LIN {X 0,Y 260.19,Z 606.09,A -85,B 0,C 180,E1 -26180.673,E2 -26180.673} C_VEL
LIN {X 0,Y 265.436,Z 608.192,A -85,B 0,C 180,E1 -26182.392,E2 -26182.392} C_VEL
LIN {X 0,Y 269.491,Z 609.865,A -85,B 0,C 180,E1 -26184.012,E2 -26184.012} C_VEL
LIN {X 0,Y 272.352,Z 611.178,A -85,B 0,C 180,E1 -26185.56,E2 -26185.56} C_VEL
LIN {X 0,Y 274.974,Z 612.087,A -85,B 0,C 180,E1 -26187.07,E2 -26187.07} C_VEL
LIN {X 0,Y 276.592,Z 612.646,A -85,B 0,C 180,E1 -26188.544,E2 -26188.544} C_VEL
LIN {X 0,Y 277.503,Z 612.825,A -85,B 0,C 180,E1 -26190,E2 -26190} C_VEL
LIN {X 0,Y 276.602,Z 612.645,A -85,B 0,C 180,E1 -26191.455,E2 -26191.455} C_VEL
LIN {X 0,Y 274.515,Z 611.947,A -85,B 0,C 180,E1 -26193.199,E2 -26193.199} C_VEL
LIN {X 0,Y 272.336,Z 611.179,A -85,B 0,C 180,E1 -26194.44,E2 -26194.44} C_VEL
LIN {X 0,Y 268.698,Z 609.555,A -85,B 0,C 180,E1 -26196.331,E2 -26196.331} C_VEL
LIN {X 0,Y 265.447,Z 608.193,A -85,B 0,C 180,E1 -26197.607,E2 -26197.607} C_VEL
LIN {X 0,Y 260.192,Z 606.091,A -85,B 0,C 180,E1 -26199.326,E2 -26199.326} C_VEL
LIN {X 0,Y 253.891,Z 603.535,A -85,B 0,C 180,E1 -26201.172,E2 -26201.172} C_VEL
LIN {X 0,Y 245.622,Z 600.226,A -85,B 0,C 180,E1 -26203.388,E2 -26203.388} C_VEL
LIN {X 0,Y 234.391,Z 595.435,A -85,B 0,C 180,E1 -26206.368,E2 -26206.368} C_VEL
LIN {X 0,Y 220.959,Z 588.75,A -85,B 0,C 180,E1 -26210.238,E2 -26210.238} C_VEL
LIN {X 0,Y 208.557,Z 580.602,A -85,B 0,C 180,E1 -26214.518,E2 -26214.518} C_VEL
LIN {X 0,Y 199.491,Z 572.681,A -85,B 0,C 180,E1 -26218.271,E2 -26218.271} C_VEL
LIN {X 0,Y 191.268,Z 563.212,A -85,B 0,C 180,E1 -26222.318,E2 -26222.318} C_VEL
LIN {X 0,Y 184.44,Z 553.289,A -85,B 0,C 180,E1 -26226.147,E2 -26226.147} C_VEL
LIN {X 0,Y 179.392,Z 544.208,A -85,B 0,C 180,E1 -26229.311,E2 -26229.311} C_VEL
LIN {X 0,Y 175.265,Z 535.205,A -85,B 0,C 180,E1 -26232.114,E2 -26232.114} C_VEL
LIN {X 0,Y 171.108,Z 524.747,A -85,B 0,C 180,E1 -26234.991,E2 -26234.991} C_VEL
LIN {X 0,Y 167.297,Z 514.145,A -85,B 0,C 180,E1 -26237.566,E2 -26237.566} C_VEL
LIN {X 0,Y 160.835,Z 495.6,A -85,B 0,C 180,E1 -26241.588,E2 -26241.588} C_VEL
LIN {X 0,Y 157.196,Z 486.8,A -85,B 0,C 180,E1 -26243.972,E2 -26243.972} C_VEL
LIN {X 0,Y 152.993,Z 478.107,A -85,B 0,C 180,E1 -26246.943,E2 -26246.943} C_VEL
LIN {X 0,Y 148.523,Z 469.896,A -85,B 0,C 180,E1 -26250.502,E2 -26250.502} C_VEL
LIN {X 0,Y 144.159,Z 462.807,A -85,B 0,C 180,E1 -26254.558,E2 -26254.558} C_VEL
LIN {X 0,Y 141.726,Z 459.081,A -85,B 0,C 180,E1 -26257.208,E2 -26257.208} C_VEL
LIN {X 0,Y 138.793,Z 454.797,A -85,B 0,C 180,E1 -26260.984,E2 -26260.984} C_VEL
LIN {X 0,Y 136.479,Z 451.612,A -85,B 0,C 180,E1 -26264.699,E2 -26264.699} C_VEL
LIN {X 0,Y 135.908,Z 450.393,A -85,B 0,C 180,E1 -26265.878,E2 -26265.878} C_VEL
LIN {X 0,Y 133.785,Z 448.176,A -85,B 0,C 180,E1 -26270.934,E2 -26270.934} C_VEL
LIN {X 0,Y 132.733,Z 445.405,A -85,B 0,C 180,E1 -26276.587,E2 -26276.587} C_VEL
LIN {X 0,Y 132.581,Z 444.946,A -85,B 0,C 180,E1 -26280.002,E2 -26280.002} C_VEL
LIN {X 0,Y 132.86,Z 445.806,A -85,B 0,C 180,E1 -26284.173,E2 -26284.173} C_VEL
LIN {X 0,Y 135.26,Z 449.966,A -85,B 0,C 180,E1 -26292.482,E2 -26292.482} C_VEL
LIN {X 0,Y 136.045,Z 450.627,A -85,B 0,C 180,E1 -26294.015,E2 -26294.015} C_VEL
LIN {X 0,Y 138.067,Z 454.011,A -85,B 0,C 180,E1 -26297.594,E2 -26297.594} C_VEL
LIN {X 0,Y 139.483,Z 455.822,A -85,B 0,C 180,E1 -26299.597,E2 -26299.597} C_VEL
LIN {X 0,Y 142.535,Z 460.338,A -85,B 0,C 180,E1 -26303.33,E2 -26303.33} C_VEL
LIN {X 0,Y 145.461,Z 464.955,A -85,B 0,C 180,E1 -26306.355,E2 -26306.355} C_VEL
LIN {X 0,Y 147.881,Z 468.942,A -85,B 0,C 180,E1 -26308.571,E2 -26308.571} C_VEL
LIN {X 0,Y 151.068,Z 476.333,A -85,B 0,C 180,E1 -26311.365,E2 -26311.365} C_VEL
LIN {X 0,Y 155.214,Z 487.342,A -85,B 0,C 180,E1 -26314.658,E2 -26314.658} C_VEL
LIN {X 0,Y 156.571,Z 491.711,A -85,B 0,C 180,E1 -26315.701,E2 -26315.701} C_VEL
LIN {X 0,Y 154.226,Z 518.872,A -85,B 0,C 180,E1 -26316.735,E2 -26316.735} C_VEL
LIN {X 0,Y 152.512,Z 529.749,A -85,B 0,C 180,E1 -26317.377,E2 -26317.377} C_VEL
LIN {X 0,Y 150.32,Z 539.537,A -85,B 0,C 180,E1 -26318.185,E2 -26318.185} C_VEL
LIN {X 0,Y 147.435,Z 549.33,A -85,B 0,C 180,E1 -26319.232,E2 -26319.232} C_VEL
LIN {X 0,Y 144.317,Z 558.091,A -85,B 0,C 180,E1 -26320.458,E2 -26320.458} C_VEL
LIN {X 0,Y 140.709,Z 566.811,A -85,B 0,C 180,E1 -26322.018,E2 -26322.018} C_VEL
LIN {X 0,Y 136.625,Z 575.317,A -85,B 0,C 180,E1 -26323.934,E2 -26323.934} C_VEL
LIN {X 0,Y 132.189,Z 583.484,A -85,B 0,C 180,E1 -26326.28,E2 -26326.28} C_VEL
LIN {X 0,Y 128.035,Z 590.426,A -85,B 0,C 180,E1 -26328.802,E2 -26328.802} C_VEL
LIN {X 0,Y 124.132,Z 596.412,A -85,B 0,C 180,E1 -26331.482,E2 -26331.482} C_VEL
LIN {X 0,Y 119.301,Z 603.383,A -85,B 0,C 180,E1 -26335.565,E2 -26335.565} C_VEL
LIN {X 0,Y 115.991,Z 608.001,A -85,B 0,C 180,E1 -26339.003,E2 -26339.003} C_VEL
LIN {X 0,Y 111.975,Z 613.094,A -85,B 0,C 180,E1 -26343.939,E2 -26343.939} C_VEL
LIN {X 0,Y 108.807,Z 617.061,A -85,B 0,C 180,E1 -26349.193,E2 -26349.193} C_VEL
LIN {X 0,Y 106.705,Z 620.004,A -85,B 0,C 180,E1 -26354.726,E2 -26354.726} C_VEL
LIN {X 0,Y 105.799,Z 621.512,A -85,B 0,C 180,E1 -26358.506,E2 -26358.506} C_VEL
LIN {X 0,Y 105.048,Z 623.051,A -85,B 0,C 180,E1 -26366.165,E2 -26366.165} C_VEL
LIN {X 0,Y 105.171,Z 623.337,A -85,B 0,C 180,E1 -26370.001,E2 -26370.001} C_VEL
LIN {X 0,Y 105.226,Z 622.446,A -85,B 0,C 180,E1 -26377.678,E2 -26377.678} C_VEL
LIN {X 0,Y 105.782,Z 621.511,A -85,B 0,C 180,E1 -26381.498,E2 -26381.498} C_VEL
LIN {X 0,Y 107.976,Z 618.15,A -85,B 0,C 180,E1 -26388.993,E2 -26388.993} C_VEL
LIN {X 0,Y 110.812,Z 614.521,A -85,B 0,C 180,E1 -26394.347,E2 -26394.347} C_VEL
LIN {X 0,Y 114.51,Z 609.787,A -85,B 0,C 180,E1 -26399.407,E2 -26399.407} C_VEL
LIN {X 0,Y 118.573,Z 604.41,A -85,B 0,C 180,E1 -26403.712,E2 -26403.712} C_VEL
LIN {X 0,Y 122.385,Z 599.035,A -85,B 0,C 180,E1 -26407.083,E2 -26407.083} C_VEL
LIN {X 0,Y 126.08,Z 593.543,A -85,B 0,C 180,E1 -26409.87,E2 -26409.87} C_VEL
LIN {X 0,Y 131.164,Z 585.33,A -85,B 0,C 180,E1 -26413.092,E2 -26413.092} C_VEL
LIN {X 0,Y 135.503,Z 577.507,A -85,B 0,C 180,E1 -26415.493,E2 -26415.493} C_VEL
LIN {X 0,Y 139.53,Z 569.429,A -85,B 0,C 180,E1 -26417.447,E2 -26417.447} C_VEL
LIN {X 0,Y 143.712,Z 559.673,A -85,B 0,C 180,E1 -26419.289,E2 -26419.289} C_VEL
LIN {X 0,Y 146.801,Z 551.287,A -85,B 0,C 180,E1 -26420.532,E2 -26420.532} C_VEL
LIN {X 0,Y 149.987,Z 540.786,A -85,B 0,C 180,E1 -26421.708,E2 -26421.708} C_VEL
LIN {X 0,Y 152.454,Z 530.424,A -85,B 0,C 180,E1 -26422.545,E2 -26422.545} C_VEL
LIN {X 0,Y 154.051,Z 520.443,A -85,B 0,C 180,E1 -26423.174,E2 -26423.174} C_VEL
LIN {X 0,Y 155.953,Z 499.799,A -85,B 0,C 180,E1 -26423.992,E2 -26423.992} C_VEL
LIN {X 0,Y 156.493,Z 491.335,A -85,B 0,C 180,E1 -26424.368,E2 -26424.368} C_VEL
LIN {X 0,Y 153.68,Z 483.124,A -85,B 0,C 180,E1 -26426.519,E2 -26426.519} C_VEL
LIN {X 0,Y 149.807,Z 473.279,A -85,B 0,C 180,E1 -26429.711,E2 -26429.711} C_VEL
LIN {X 0,Y 147.096,Z 467.508,A -85,B 0,C 180,E1 -26432.137,E2 -26432.137} C_VEL
LIN {X 0,Y 143.603,Z 462.012,A -85,B 0,C 180,E1 -26435.513,E2 -26435.513} C_VEL
LIN {X 0,Y 141.546,Z 458.883,A -85,B 0,C 180,E1 -26437.797,E2 -26437.797} C_VEL
LIN {X 0,Y 138.866,Z 454.87,A -85,B 0,C 180,E1 -26441.271,E2 -26441.271} C_VEL
LIN {X 0,Y 137.213,Z 452.876,A -85,B 0,C 180,E1 -26443.757,E2 -26443.757} C_VEL
LIN {X 0,Y 136.228,Z 452.315,A -85,B 0,C 180,E1 -26445.339,E2 -26445.339} C_VEL
LIN {X 0,Y 134.55,Z 453.443,A -85,B 0,C 180,E1 -26448.044,E2 -26448.044} C_VEL
LIN {X 0,Y 133.132,Z 454.874,A -85,B 0,C 180,E1 -26450.839,E2 -26450.839} C_VEL
LIN {X 0,Y 132.552,Z 454.745,A -85,B 0,C 180,E1 -26452.56,E2 -26452.56} C_VEL
LIN {X 0,Y 131.864,Z 452.504,A -85,B 0,C 180,E1 -26456.943,E2 -26456.943} C_VEL
LIN {X 0,Y 131.714,Z 452.009,A -85,B 0,C 180,E1 -26459.998,E2 -26459.998} C_VEL
LIN {X 0,Y 131.937,Z 452.812,A -85,B 0,C 180,E1 -26464.199,E2 -26464.199} C_VEL
LIN {X 0,Y 134.017,Z 456.758,A -85,B 0,C 180,E1 -26472.107,E2 -26472.107} C_VEL
LIN {X 0,Y 134.831,Z 457.672,A -85,B 0,C 180,E1 -26473.852,E2 -26473.852} C_VEL
LIN {X 0,Y 137.166,Z 461.404,A -85,B 0,C 180,E1 -26478.049,E2 -26478.049} C_VEL
LIN {X 0,Y 138.154,Z 462.984,A -85,B 0,C 180,E1 -26479.524,E2 -26479.524} C_VEL
LIN {X 0,Y 140.751,Z 466.949,A -85,B 0,C 180,E1 -26482.861,E2 -26482.861} C_VEL
LIN {X 0,Y 144.345,Z 472.817,A -85,B 0,C 180,E1 -26486.712,E2 -26486.712} C_VEL
LIN {X 0,Y 148.947,Z 481.421,A -85,B 0,C 180,E1 -26490.871,E2 -26490.871} C_VEL
LIN {X 0,Y 153.195,Z 490.333,A -85,B 0,C 180,E1 -26494.191,E2 -26494.191} C_VEL
LIN {X 0,Y 156.819,Z 499.361,A -85,B 0,C 180,E1 -26496.792,E2 -26496.792} C_VEL
LIN {X 0,Y 161.027,Z 512.279,A -85,B 0,C 180,E1 -26499.765,E2 -26499.765} C_VEL
LIN {X 0,Y 163.994,Z 521.801,A -85,B 0,C 180,E1 -26502.035,E2 -26502.035} C_VEL
LIN {X 0,Y 166.737,Z 529.994,A -85,B 0,C 180,E1 -26504.229,E2 -26504.229} C_VEL
LIN {X 0,Y 170.461,Z 540.108,A -85,B 0,C 180,E1 -26507.281,E2 -26507.281} C_VEL
LIN {X 0,Y 174.845,Z 550.091,A -85,B 0,C 180,E1 -26510.691,E2 -26510.691} C_VEL
LIN {X 0,Y 179.722,Z 558.93,A -85,B 0,C 180,E1 -26514.085,E2 -26514.085} C_VEL
LIN {X 0,Y 184.9,Z 566.539,A -85,B 0,C 180,E1 -26517.284,E2 -26517.284} C_VEL
LIN {X 0,Y 192.281,Z 575.252,A -85,B 0,C 180,E1 -26521.306,E2 -26521.306} C_VEL
LIN {X 0,Y 201.115,Z 583.076,A -85,B 0,C 180,E1 -26525.306,E2 -26525.306} C_VEL
LIN {X 0,Y 210.822,Z 589.611,A -85,B 0,C 180,E1 -26528.97,E2 -26528.97} C_VEL
LIN {X 0,Y 221.311,Z 595.053,A -85,B 0,C 180,E1 -26532.301,E2 -26532.301} C_VEL
LIN {X 0,Y 235.105,Z 600.84,A -85,B 0,C 180,E1 -26536.164,E2 -26536.164} C_VEL
LIN {X 0,Y 246.771,Z 605.064,A -85,B 0,C 180,E1 -26539.276,E2 -26539.276} C_VEL
LIN {X 0,Y 250.405,Z 606.363,A -85,B 0,C 180,E1 -26540.305,E2 -26540.305} C_VEL
LIN {X 0,Y 256.397,Z 608.44,A -85,B 0,C 180,E1 -26542.122,E2 -26542.122} C_VEL
LIN {X 0,Y 261.473,Z 610.236,A -85,B 0,C 180,E1 -26543.981,E2 -26543.981} C_VEL
LIN {X 0,Y 264.49,Z 611.396,A -85,B 0,C 180,E1 -26545.427,E2 -26545.427} C_VEL
LIN {X 0,Y 267.412,Z 612.332,A -85,B 0,C 180,E1 -26547.055,E2 -26547.055} C_VEL
LIN {X 0,Y 269.266,Z 612.848,A -85,B 0,C 180,E1 -26548.504,E2 -26548.504} C_VEL
LIN {X 0,Y 270.336,Z 613.022,A -85,B 0,C 180,E1 -26550,E2 -26550} C_VEL
LIN {X 0,Y 269.274,Z 612.847,A -85,B 0,C 180,E1 -26551.495,E2 -26551.495} C_VEL
LIN {X 0,Y 267.273,Z 612.298,A -85,B 0,C 180,E1 -26553.014,E2 -26553.014} C_VEL
LIN {X 0,Y 264.455,Z 611.398,A -85,B 0,C 180,E1 -26554.572,E2 -26554.572} C_VEL
LIN {X 0,Y 261.051,Z 610.097,A -85,B 0,C 180,E1 -26556.182,E2 -26556.182} C_VEL
LIN {X 0,Y 255.575,Z 608.153,A -85,B 0,C 180,E1 -26558.134,E2 -26558.134} C_VEL
LIN {X 0,Y 249.687,Z 606.114,A -85,B 0,C 180,E1 -26559.892,E2 -26559.892} C_VEL
LIN {X 0,Y 243.257,Z 603.834,A -85,B 0,C 180,E1 -26561.667,E2 -26561.667} C_VEL
LIN {X 0,Y 232.366,Z 599.799,A -85,B 0,C 180,E1 -26564.572,E2 -26564.572} C_VEL
LIN {X 0,Y 217.485,Z 593.257,A -85,B 0,C 180,E1 -26568.853,E2 -26568.853} C_VEL
LIN {X 0,Y 205.887,Z 586.508,A -85,B 0,C 180,E1 -26572.835,E2 -26572.835} C_VEL
LIN {X 0,Y 195.482,Z 578.371,A -85,B 0,C 180,E1 -26577.154,E2 -26577.154} C_VEL
LIN {X 0,Y 188.219,Z 570.743,A -85,B 0,C 180,E1 -26580.82,E2 -26580.82} C_VEL
LIN {X 0,Y 181.609,Z 561.932,A -85,B 0,C 180,E1 -26584.682,E2 -26584.682} C_VEL
LIN {X 0,Y 176.652,Z 553.661,A -85,B 0,C 180,E1 -26587.988,E2 -26587.988} C_VEL
LIN {X 0,Y 172.518,Z 545.013,A -85,B 0,C 180,E1 -26591.093,E2 -26591.093} C_VEL
LIN {X 0,Y 168.776,Z 535.798,A -85,B 0,C 180,E1 -26594.078,E2 -26594.078} C_VEL
LIN {X 0,Y 164.91,Z 524.737,A -85,B 0,C 180,E1 -26597.22,E2 -26597.22} C_VEL
LIN {X 0,Y 161.46,Z 513.632,A -85,B 0,C 180,E1 -26599.956,E2 -26599.956} C_VEL
LIN {X 0,Y 157.032,Z 499.987,A -85,B 0,C 180,E1 -26603.056,E2 -26603.056} C_VEL
LIN {X 0,Y 153.632,Z 491.36,A -85,B 0,C 180,E1 -26605.484,E2 -26605.484} C_VEL
LIN {X 0,Y 149.79,Z 483.094,A -85,B 0,C 180,E1 -26608.438,E2 -26608.438} C_VEL
LIN {X 0,Y 145.811,Z 475.456,A -85,B 0,C 180,E1 -26611.883,E2 -26611.883} C_VEL
LIN {X 0,Y 142.008,Z 468.949,A -85,B 0,C 180,E1 -26615.71,E2 -26615.71} C_VEL
LIN {X 0,Y 139.706,Z 465.279,A -85,B 0,C 180,E1 -26618.418,E2 -26618.418} C_VEL
LIN {X 0,Y 137.263,Z 461.492,A -85,B 0,C 180,E1 -26621.812,E2 -26621.812} C_VEL
LIN {X 0,Y 134.87,Z 457.777,A -85,B 0,C 180,E1 -26626.056,E2 -26626.056} C_VEL
LIN {X 0,Y 134.235,Z 456.928,A -85,B 0,C 180,E1 -26627.417,E2 -26627.417} C_VEL
LIN {X 0,Y 132.192,Z 453.826,A -85,B 0,C 180,E1 -26633.898,E2 -26633.898} C_VEL
LIN {X 0,Y 131.829,Z 452.405,A -85,B 0,C 180,E1 -26636.946,E2 -26636.946} C_VEL
LIN {X 0,Y 131.715,Z 452.001,A -85,B 0,C 180,E1 -26640.002,E2 -26640.002} C_VEL
LIN {X 0,Y 131.947,Z 452.868,A -85,B 0,C 180,E1 -26643.915,E2 -26643.915} C_VEL
LIN {X 0,Y 134.184,Z 456.923,A -85,B 0,C 180,E1 -26652.095,E2 -26652.095} C_VEL
LIN {X 0,Y 134.816,Z 457.622,A -85,B 0,C 180,E1 -26653.429,E2 -26653.429} C_VEL
LIN {X 0,Y 137.201,Z 461.408,A -85,B 0,C 180,E1 -26657.708,E2 -26657.708} C_VEL
LIN {X 0,Y 140.492,Z 466.502,A -85,B 0,C 180,E1 -26662.161,E2 -26662.161} C_VEL
LIN {X 0,Y 144.393,Z 472.874,A -85,B 0,C 180,E1 -26666.37,E2 -26666.37} C_VEL
LIN {X 0,Y 146.946,Z 478.613,A -85,B 0,C 180,E1 -26668.867,E2 -26668.867} C_VEL
LIN {X 0,Y 151.241,Z 490.424,A -85,B 0,C 180,E1 -26672.699,E2 -26672.699} C_VEL
LIN {X 0,Y 152.325,Z 493.979,A -85,B 0,C 180,E1 -26673.62,E2 -26673.62} C_VEL
LIN {X 0,Y 150.039,Z 519.059,A -85,B 0,C 180,E1 -26674.58,E2 -26674.58} C_VEL
LIN {X 0,Y 148.058,Z 530.895,A -85,B 0,C 180,E1 -26675.289,E2 -26675.289} C_VEL
LIN {X 0,Y 144.725,Z 544.21,A -85,B 0,C 180,E1 -26676.46,E2 -26676.46} C_VEL
LIN {X 0,Y 140.461,Z 556.307,A -85,B 0,C 180,E1 -26677.998,E2 -26677.998} C_VEL
LIN {X 0,Y 136.686,Z 565.304,A -85,B 0,C 180,E1 -26679.536,E2 -26679.536} C_VEL
LIN {X 0,Y 132.397,Z 574.024,A -85,B 0,C 180,E1 -26681.429,E2 -26681.429} C_VEL
LIN {X 0,Y 128.294,Z 581.44,A -85,B 0,C 180,E1 -26683.463,E2 -26683.463} C_VEL
LIN {X 0,Y 122.78,Z 590.231,A -85,B 0,C 180,E1 -26686.618,E2 -26686.618} C_VEL
LIN {X 0,Y 118.641,Z 596.217,A -85,B 0,C 180,E1 -26689.339,E2 -26689.339} C_VEL
LIN {X 0,Y 113.961,Z 602.585,A -85,B 0,C 180,E1 -26693.098,E2 -26693.098} C_VEL
LIN {X 0,Y 109.952,Z 607.805,A -85,B 0,C 180,E1 -26697.093,E2 -26697.093} C_VEL
LIN {X 0,Y 105.614,Z 612.899,A -85,B 0,C 180,E1 -26702.239,E2 -26702.239} C_VEL
LIN {X 0,Y 102.184,Z 616.865,A -85,B 0,C 180,E1 -26707.774,E2 -26707.774} C_VEL
LIN {X 0,Y 99.83,Z 619.808,A -85,B 0,C 180,E1 -26713.646,E2 -26713.646} C_VEL
LIN {X 0,Y 98.814,Z 621.316,A -85,B 0,C 180,E1 -26717.681,E2 -26717.681} C_VEL
LIN {X 0,Y 97.954,Z 622.855,A -85,B 0,C 180,E1 -26725.887,E2 -26725.887} C_VEL
LIN {X 0,Y 98.077,Z 623.142,A -85,B 0,C 180,E1 -26730.001,E2 -26730.001} C_VEL
LIN {X 0,Y 98.183,Z 622.251,A -85,B 0,C 180,E1 -26738.232,E2 -26738.232} C_VEL
LIN {X 0,Y 98.8,Z 621.315,A -85,B 0,C 180,E1 -26742.323,E2 -26742.323} C_VEL
LIN {X 0,Y 101.249,Z 617.954,A -85,B 0,C 180,E1 -26750.309,E2 -26750.309} C_VEL
LIN {X 0,Y 104.353,Z 614.325,A -85,B 0,C 180,E1 -26755.962,E2 -26755.962} C_VEL
LIN {X 0,Y 108.37,Z 609.592,A -85,B 0,C 180,E1 -26761.254,E2 -26761.254} C_VEL
LIN {X 0,Y 113.446,Z 603.323,A -85,B 0,C 180,E1 -26766.353,E2 -26766.353} C_VEL
LIN {X 0,Y 118.681,Z 596.215,A -85,B 0,C 180,E1 -26770.647,E2 -26770.647} C_VEL
LIN {X 0,Y 124.957,Z 586.984,A -85,B 0,C 180,E1 -26774.672,E2 -26774.672} C_VEL
LIN {X 0,Y 130.624,Z 577.312,A -85,B 0,C 180,E1 -26777.715,E2 -26777.715} C_VEL
LIN {X 0,Y 134.824,Z 569.233,A -85,B 0,C 180,E1 -26779.673,E2 -26779.673} C_VEL
LIN {X 0,Y 139.19,Z 559.478,A -85,B 0,C 180,E1 -26781.502,E2 -26781.502} C_VEL
LIN {X 0,Y 142.404,Z 551.093,A -85,B 0,C 180,E1 -26782.732,E2 -26782.732} C_VEL
LIN {X 0,Y 145.704,Z 540.592,A -85,B 0,C 180,E1 -26783.895,E2 -26783.895} C_VEL
LIN {X 0,Y 148.238,Z 530.23,A -85,B 0,C 180,E1 -26784.727,E2 -26784.727} C_VEL
LIN {X 0,Y 149.952,Z 519.805,A -85,B 0,C 180,E1 -26785.369,E2 -26785.369} C_VEL
LIN {X 0,Y 151.983,Z 498.522,A -85,B 0,C 180,E1 -26786.195,E2 -26786.195} C_VEL
LIN {X 0,Y 152.232,Z 493.691,A -85,B 0,C 180,E1 -26786.456,E2 -26786.456} C_VEL
LIN {X 0,Y 149.701,Z 486.086,A -85,B 0,C 180,E1 -26788.611,E2 -26788.611} C_VEL
LIN {X 0,Y 146.364,Z 477.146,A -85,B 0,C 180,E1 -26791.693,E2 -26791.693} C_VEL
LIN {X 0,Y 144.229,Z 472.588,A -85,B 0,C 180,E1 -26793.792,E2 -26793.792} C_VEL
LIN {X 0,Y 140.032,Z 465.681,A -85,B 0,C 180,E1 -26798.411,E2 -26798.411} C_VEL
LIN {X 0,Y 137.205,Z 461.375,A -85,B 0,C 180,E1 -26802.292,E2 -26802.292} C_VEL
LIN {X 0,Y 134.792,Z 457.59,A -85,B 0,C 180,E1 -26806.621,E2 -26806.621} C_VEL
LIN {X 0,Y 132.552,Z 454.745,A -85,B 0,C 180,E1 -26812.56,E2 -26812.56} C_VEL
LIN {X 0,Y 131.946,Z 454.341,A -85,B 0,C 180,E1 -26815.109,E2 -26815.109} C_VEL
LIN {X 0,Y 131.459,Z 455.108,A -85,B 0,C 180,E1 -26817.676,E2 -26817.676} C_VEL
LIN {X 0,Y 131.04,Z 458.564,A -85,B 0,C 180,E1 -26822.766,E2 -26822.766} C_VEL
LIN {X 0,Y 131.316,Z 461.049,A -85,B 0,C 180,E1 -26826.168,E2 -26826.168} C_VEL
LIN {X 0,Y 133.158,Z 463.912,A -85,B 0,C 180,E1 -26832.186,E2 -26832.186} C_VEL
LIN {X 0,Y 133.638,Z 464.692,A -85,B 0,C 180,E1 -26833.301,E2 -26833.301} C_VEL
LIN {X 0,Y 136.276,Z 469.035,A -85,B 0,C 180,E1 -26838.171,E2 -26838.171} C_VEL
LIN {X 0,Y 138.819,Z 473.253,A -85,B 0,C 180,E1 -26841.756,E2 -26841.756} C_VEL
LIN {X 0,Y 142.055,Z 478.83,A -85,B 0,C 180,E1 -26845.502,E2 -26845.502} C_VEL
LIN {X 0,Y 146.249,Z 487.15,A -85,B 0,C 180,E1 -26849.606,E2 -26849.606} C_VEL
LIN {X 0,Y 150.02,Z 495.572,A -85,B 0,C 180,E1 -26852.808,E2 -26852.808} C_VEL
LIN {X 0,Y 153.323,Z 504.298,A -85,B 0,C 180,E1 -26855.389,E2 -26855.389} C_VEL
LIN {X 0,Y 157.441,Z 518.413,A -85,B 0,C 180,E1 -26858.779,E2 -26858.779} C_VEL
LIN {X 0,Y 160.7,Z 530.237,A -85,B 0,C 180,E1 -26861.972,E2 -26861.972} C_VEL
LIN {X 0,Y 163.942,Z 540.571,A -85,B 0,C 180,E1 -26865.188,E2 -26865.188} C_VEL
LIN {X 0,Y 167.18,Z 549.175,A -85,B 0,C 180,E1 -26868.202,E2 -26868.202} C_VEL
LIN {X 0,Y 170.885,Z 557.426,A -85,B 0,C 180,E1 -26871.388,E2 -26871.388} C_VEL
LIN {X 0,Y 176.487,Z 566.964,A -85,B 0,C 180,E1 -26875.562,E2 -26875.562} C_VEL
LIN {X 0,Y 183.143,Z 575.615,A -85,B 0,C 180,E1 -26879.758,E2 -26879.758} C_VEL
LIN {X 0,Y 190.735,Z 583.108,A -85,B 0,C 180,E1 -26883.758,E2 -26883.758} C_VEL
LIN {X 0,Y 198.359,Z 588.846,A -85,B 0,C 180,E1 -26887.098,E2 -26887.098} C_VEL
LIN {X 0,Y 208.377,Z 594.647,A -85,B 0,C 180,E1 -26890.795,E2 -26890.795} C_VEL
LIN {X 0,Y 219.164,Z 599.447,A -85,B 0,C 180,E1 -26894.154,E2 -26894.154} C_VEL
LIN {X 0,Y 232.135,Z 604.145,A -85,B 0,C 180,E1 -26897.764,E2 -26897.764} C_VEL
LIN {X 0,Y 242.265,Z 607.327,A -85,B 0,C 180,E1 -26900.506,E2 -26900.506} C_VEL
LIN {X 0,Y 248.229,Z 609.15,A -85,B 0,C 180,E1 -26902.274,E2 -26902.274} C_VEL
LIN {X 0,Y 254.245,Z 610.938,A -85,B 0,C 180,E1 -26904.336,E2 -26904.336} C_VEL
LIN {X 0,Y 256.401,Z 611.621,A -85,B 0,C 180,E1 -26905.283,E2 -26905.283} C_VEL
LIN {X 0,Y 260.315,Z 612.713,A -85,B 0,C 180,E1 -26907.324,E2 -26907.324} C_VEL
LIN {X 0,Y 261.846,Z 613.051,A -85,B 0,C 180,E1 -26908.462,E2 -26908.462} C_VEL
LIN {X 0,Y 263.144,Z 613.219,A -85,B 0,C 180,E1 -26910,E2 -26910} C_VEL
LIN {X 0,Y 261.85,Z 613.051,A -85,B 0,C 180,E1 -26911.538,E2 -26911.538} C_VEL
LIN {X 0,Y 259.5,Z 612.51,A -85,B 0,C 180,E1 -26913.104,E2 -26913.104} C_VEL
LIN {X 0,Y 256.384,Z 611.622,A -85,B 0,C 180,E1 -26914.717,E2 -26914.717} C_VEL
LIN {X 0,Y 254.244,Z 610.938,A -85,B 0,C 180,E1 -26915.663,E2 -26915.663} C_VEL
LIN {X 0,Y 248.228,Z 609.152,A -85,B 0,C 180,E1 -26917.724,E2 -26917.724} C_VEL
LIN {X 0,Y 239.985,Z 606.656,A -85,B 0,C 180,E1 -26920.119,E2 -26920.119} C_VEL
LIN {X 0,Y 227.617,Z 602.646,A -85,B 0,C 180,E1 -26923.447,E2 -26923.447} C_VEL
LIN {X 0,Y 213.674,Z 597.156,A -85,B 0,C 180,E1 -26927.479,E2 -26927.479} C_VEL
LIN {X 0,Y 203.261,Z 591.87,A -85,B 0,C 180,E1 -26931.007,E2 -26931.007} C_VEL
LIN {X 0,Y 193.68,Z 585.491,A -85,B 0,C 180,E1 -26934.886,E2 -26934.886} C_VEL
LIN {X 0,Y 186.116,Z 578.761,A -85,B 0,C 180,E1 -26938.607,E2 -26938.607} C_VEL
LIN {X 0,Y 179.297,Z 570.903,A -85,B 0,C 180,E1 -26942.573,E2 -26942.573} C_VEL
LIN {X 0,Y 174.066,Z 563.15,A -85,B 0,C 180,E1 -26946.149,E2 -26946.149} C_VEL
LIN {X 0,Y 169.191,Z 553.993,A -85,B 0,C 180,E1 -26949.97,E2 -26949.97} C_VEL
LIN {X 0,Y 165.131,Z 543.95,A -85,B 0,C 180,E1 -26953.656,E2 -26953.656} C_VEL
LIN {X 0,Y 162.529,Z 536.191,A -85,B 0,C 180,E1 -26956.224,E2 -26956.224} C_VEL
LIN {X 0,Y 159.37,Z 525.643,A -85,B 0,C 180,E1 -26959.322,E2 -26959.322} C_VEL
LIN {X 0,Y 156.219,Z 513.867,A -85,B 0,C 180,E1 -26962.3,E2 -26962.3} C_VEL
LIN {X 0,Y 152.83,Z 502.981,A -85,B 0,C 180,E1 -26964.979,E2 -26964.979} C_VEL
LIN {X 0,Y 149.819,Z 495.068,A -85,B 0,C 180,E1 -26967.356,E2 -26967.356} C_VEL
LIN {X 0,Y 145.899,Z 486.413,A -85,B 0,C 180,E1 -26970.712,E2 -26970.712} C_VEL
LIN {X 0,Y 142.242,Z 479.268,A -85,B 0,C 180,E1 -26974.288,E2 -26974.288} C_VEL
LIN {X 0,Y 139.449,Z 474.364,A -85,B 0,C 180,E1 -26977.451,E2 -26977.451} C_VEL
LIN {X 0,Y 137.601,Z 471.28,A -85,B 0,C 180,E1 -26979.86,E2 -26979.86} C_VEL
LIN {X 0,Y 135.58,Z 467.946,A -85,B 0,C 180,E1 -26982.952,E2 -26982.952} C_VEL
LIN {X 0,Y 133.161,Z 463.888,A -85,B 0,C 180,E1 -26987.814,E2 -26987.814} C_VEL
LIN {X 0,Y 131.213,Z 460.778,A -85,B 0,C 180,E1 -26994.431,E2 -26994.431} C_VEL
LIN {X 0,Y 130.904,Z 459.324,A -85,B 0,C 180,E1 -26997.694,E2 -26997.694} C_VEL
LIN {X 0,Y 130.854,Z 459.153,A -85,B 0,C 180,E1 -27000.771,E2 -27000.771} C_VEL
LIN {X 0,Y 131.035,Z 459.937,A -85,B 0,C 180,E1 -27003.653,E2 -27003.653} C_VEL
LIN {X 0,Y 133.16,Z 463.908,A -85,B 0,C 180,E1 -27011.803,E2 -27011.803} C_VEL
LIN {X 0,Y 133.689,Z 464.804,A -85,B 0,C 180,E1 -27013.035,E2 -27013.035} C_VEL
LIN {X 0,Y 136.246,Z 468.996,A -85,B 0,C 180,E1 -27017.74,E2 -27017.74} C_VEL
LIN {X 0,Y 138.746,Z 473.084,A -85,B 0,C 180,E1 -27021.269,E2 -27021.269} C_VEL
LIN {X 0,Y 142.222,Z 479.165,A -85,B 0,C 180,E1 -27025.296,E2 -27025.296} C_VEL
LIN {X 0,Y 144.255,Z 484.19,A -85,B 0,C 180,E1 -27027.473,E2 -27027.473} C_VEL
LIN {X 0,Y 148.011,Z 495.377,A -85,B 0,C 180,E1 -27031.167,E2 -27031.167} C_VEL
LIN {X 0,Y 148.299,Z 496.595,A -85,B 0,C 180,E1 -27031.46,E2 -27031.46} C_VEL
LIN {X 0,Y 146.028,Z 519.616,A -85,B 0,C 180,E1 -27032.322,E2 -27032.322} C_VEL
LIN {X 0,Y 143.791,Z 532.12,A -85,B 0,C 180,E1 -27033.076,E2 -27033.076} C_VEL
LIN {X 0,Y 140.25,Z 545.005,A -85,B 0,C 180,E1 -27034.229,E2 -27034.229} C_VEL
LIN {X 0,Y 136.205,Z 556.112,A -85,B 0,C 180,E1 -27035.644,E2 -27035.644} C_VEL
LIN {X 0,Y 132.277,Z 565.109,A -85,B 0,C 180,E1 -27037.161,E2 -27037.161} C_VEL
LIN {X 0,Y 127.81,Z 573.829,A -85,B 0,C 180,E1 -27039.042,E2 -27039.042} C_VEL
LIN {X 0,Y 123.52,Z 581.245,A -85,B 0,C 180,E1 -27041.074,E2 -27041.074} C_VEL
LIN {X 0,Y 117.702,Z 590.035,A -85,B 0,C 180,E1 -27044.234,E2 -27044.234} C_VEL
LIN {X 0,Y 113.341,Z 596.021,A -85,B 0,C 180,E1 -27046.996,E2 -27046.996} C_VEL
LIN {X 0,Y 108.452,Z 602.26,A -85,B 0,C 180,E1 -27050.738,E2 -27050.738} C_VEL
LIN {X 0,Y 104.032,Z 607.609,A -85,B 0,C 180,E1 -27054.956,E2 -27054.956} C_VEL
LIN {X 0,Y 99.345,Z 612.702,A -85,B 0,C 180,E1 -27060.319,E2 -27060.319} C_VEL
LIN {X 0,Y 95.611,Z 616.669,A -85,B 0,C 180,E1 -27066.155,E2 -27066.155} C_VEL
LIN {X 0,Y 93.005,Z 619.612,A -85,B 0,C 180,E1 -27072.408,E2 -27072.408} C_VEL
LIN {X 0,Y 91.864,Z 621.12,A -85,B 0,C 180,E1 -27076.733,E2 -27076.733} C_VEL
LIN {X 0,Y 90.882,Z 622.66,A -85,B 0,C 180,E1 -27085.566,E2 -27085.566} C_VEL
LIN {X 0,Y 90.976,Z 622.947,A -85,B 0,C 180,E1 -27090.001,E2 -27090.001} C_VEL
LIN {X 0,Y 91.144,Z 622.055,A -85,B 0,C 180,E1 -27098.873,E2 -27098.873} C_VEL
LIN {X 0,Y 91.853,Z 621.119,A -85,B 0,C 180,E1 -27103.271,E2 -27103.271} C_VEL
LIN {X 0,Y 94.588,Z 617.758,A -85,B 0,C 180,E1 -27111.81,E2 -27111.81} C_VEL
LIN {X 0,Y 97.992,Z 614.129,A -85,B 0,C 180,E1 -27117.788,E2 -27117.788} C_VEL
LIN {X 0,Y 102.358,Z 609.396,A -85,B 0,C 180,E1 -27123.319,E2 -27123.319} C_VEL
LIN {X 0,Y 105.717,Z 605.609,A -85,B 0,C 180,E1 -27126.75,E2 -27126.75} C_VEL
LIN {X 0,Y 110.343,Z 599.954,A -85,B 0,C 180,E1 -27130.757,E2 -27130.757} C_VEL
LIN {X 0,Y 115.512,Z 593.152,A -85,B 0,C 180,E1 -27134.402,E2 -27134.402} C_VEL
LIN {X 0,Y 121.162,Z 584.939,A -85,B 0,C 180,E1 -27137.695,E2 -27137.695} C_VEL
LIN {X 0,Y 125.958,Z 577.117,A -85,B 0,C 180,E1 -27140.104,E2 -27140.104} C_VEL
LIN {X 0,Y 130.343,Z 569.038,A -85,B 0,C 180,E1 -27142.052,E2 -27142.052} C_VEL
LIN {X 0,Y 134.883,Z 559.283,A -85,B 0,C 180,E1 -27143.864,E2 -27143.864} C_VEL
LIN {X 0,Y 138.232,Z 550.898,A -85,B 0,C 180,E1 -27145.068,E2 -27145.068} C_VEL
LIN {X 0,Y 141.647,Z 540.397,A -85,B 0,C 180,E1 -27146.209,E2 -27146.209} C_VEL
LIN {X 0,Y 144.347,Z 529.607,A -85,B 0,C 180,E1 -27147.052,E2 -27147.052} C_VEL
LIN {X 0,Y 146.055,Z 519.507,A -85,B 0,C 180,E1 -27147.662,E2 -27147.662} C_VEL
LIN {X 0,Y 148.279,Z 496.363,A -85,B 0,C 180,E1 -27148.574,E2 -27148.574} C_VEL
LIN {X 0,Y 145.207,Z 486.884,A -85,B 0,C 180,E1 -27151.545,E2 -27151.545} C_VEL
LIN {X 0,Y 142.388,Z 479.48,A -85,B 0,C 180,E1 -27154.528,E2 -27154.528} C_VEL
LIN {X 0,Y 139.279,Z 474.039,A -85,B 0,C 180,E1 -27158.051,E2 -27158.051} C_VEL
LIN {X 0,Y 137.75,Z 471.468,A -85,B 0,C 180,E1 -27160.049,E2 -27160.049} C_VEL
LIN {X 0,Y 135.53,Z 467.844,A -85,B 0,C 180,E1 -27163.427,E2 -27163.427} C_VEL
LIN {X 0,Y 133.33,Z 464.034,A -85,B 0,C 180,E1 -27167.826,E2 -27167.826} C_VEL
LIN {X 0,Y 131.168,Z 460.508,A -85,B 0,C 180,E1 -27175.196,E2 -27175.196} C_VEL
LIN {X 0,Y 130.928,Z 459.417,A -85,B 0,C 180,E1 -27177.691,E2 -27177.691} C_VEL
LIN {X 0,Y 130.847,Z 459.068,A -85,B 0,C 180,E1 -27179.998,E2 -27179.998} C_VEL
LIN {X 0,Y 131.019,Z 459.822,A -85,B 0,C 180,E1 -27183.843,E2 -27183.843} C_VEL
LIN {X 0,Y 131.316,Z 461.049,A -85,B 0,C 180,E1 -27186.168,E2 -27186.168} C_VEL
LIN {X 0,Y 131.748,Z 463.172,A -85,B 0,C 180,E1 -27188.57,E2 -27188.57} C_VEL
LIN {X 0,Y 132.646,Z 468.233,A -85,B 0,C 180,E1 -27192.248,E2 -27192.248} C_VEL
LIN {X 0,Y 133.666,Z 472.672,A -85,B 0,C 180,E1 -27195.086,E2 -27195.086} C_VEL
LIN {X 0,Y 135.181,Z 476.509,A -85,B 0,C 180,E1 -27198.001,E2 -27198.001} C_VEL
LIN {X 0,Y 137.1,Z 479.848,A -85,B 0,C 180,E1 -27200.839,E2 -27200.839} C_VEL
LIN {X 0,Y 139.859,Z 484.951,A -85,B 0,C 180,E1 -27204.293,E2 -27204.293} C_VEL
LIN {X 0,Y 143.496,Z 492.575,A -85,B 0,C 180,E1 -27208.166,E2 -27208.166} C_VEL
LIN {X 0,Y 146.925,Z 500.742,A -85,B 0,C 180,E1 -27211.352,E2 -27211.352} C_VEL
LIN {X 0,Y 149.807,Z 509.017,A -85,B 0,C 180,E1 -27213.854,E2 -27213.854} C_VEL
LIN {X 0,Y 152.945,Z 521.511,A -85,B 0,C 180,E1 -27217.091,E2 -27217.091} C_VEL
LIN {X 0,Y 155.375,Z 531.969,A -85,B 0,C 180,E1 -27220.045,E2 -27220.045} C_VEL
LIN {X 0,Y 157.765,Z 540.915,A -85,B 0,C 180,E1 -27222.938,E2 -27222.938} C_VEL
LIN {X 0,Y 160.568,Z 550.054,A -85,B 0,C 180,E1 -27226.232,E2 -27226.232} C_VEL
LIN {X 0,Y 164.228,Z 559.451,A -85,B 0,C 180,E1 -27230.065,E2 -27230.065} C_VEL
LIN {X 0,Y 168.35,Z 567.323,A -85,B 0,C 180,E1 -27233.672,E2 -27233.672} C_VEL
LIN {X 0,Y 174.123,Z 575.731,A -85,B 0,C 180,E1 -27237.95,E2 -27237.95} C_VEL
LIN {X 0,Y 181.062,Z 583.399,A -85,B 0,C 180,E1 -27242.239,E2 -27242.239} C_VEL
LIN {X 0,Y 189.328,Z 590.065,A -85,B 0,C 180,E1 -27246.371,E2 -27246.371} C_VEL
LIN {X 0,Y 198.166,Z 595.446,A -85,B 0,C 180,E1 -27250.019,E2 -27250.019} C_VEL
LIN {X 0,Y 211.526,Z 601.298,A -85,B 0,C 180,E1 -27254.474,E2 -27254.474} C_VEL
LIN {X 0,Y 222.93,Z 605.185,A -85,B 0,C 180,E1 -27257.762,E2 -27257.762} C_VEL
LIN {X 0,Y 228.985,Z 606.963,A -85,B 0,C 180,E1 -27259.388,E2 -27259.388} C_VEL
LIN {X 0,Y 236.604,Z 608.979,A -85,B 0,C 180,E1 -27261.459,E2 -27261.459} C_VEL
LIN {X 0,Y 242.941,Z 610.592,A -85,B 0,C 180,E1 -27263.355,E2 -27263.355} C_VEL
LIN {X 0,Y 248.097,Z 611.851,A -85,B 0,C 180,E1 -27265.125,E2 -27265.125} C_VEL
LIN {X 0,Y 253.219,Z 613.043,A -85,B 0,C 180,E1 -27267.632,E2 -27267.632} C_VEL
LIN {X 0,Y 254.369,Z 613.255,A -85,B 0,C 180,E1 -27268.416,E2 -27268.416} C_VEL
LIN {X 0,Y 255.921,Z 613.418,A -85,B 0,C 180,E1 -27270,E2 -27270} C_VEL
LIN {X 0,Y 254.365,Z 613.255,A -85,B 0,C 180,E1 -27271.583,E2 -27271.583} C_VEL
LIN {X 0,Y 253.217,Z 613.047,A -85,B 0,C 180,E1 -27272.356,E2 -27272.356} C_VEL
LIN {X 0,Y 248.096,Z 611.852,A -85,B 0,C 180,E1 -27274.875,E2 -27274.875} C_VEL
LIN {X 0,Y 240.893,Z 610.105,A -85,B 0,C 180,E1 -27277.287,E2 -27277.287} C_VEL
LIN {X 0,Y 234.829,Z 608.509,A -85,B 0,C 180,E1 -27279.029,E2 -27279.029} C_VEL
LIN {X 0,Y 228.834,Z 606.92,A -85,B 0,C 180,E1 -27280.651,E2 -27280.651} C_VEL
LIN {X 0,Y 217.163,Z 603.358,A -85,B 0,C 180,E1 -27283.865,E2 -27283.865} C_VEL
LIN {X 0,Y 203.409,Z 598.002,A -85,B 0,C 180,E1 -27288.116,E2 -27288.116} C_VEL
LIN {X 0,Y 193.761,Z 592.955,A -85,B 0,C 180,E1 -27291.732,E2 -27291.732} C_VEL
LIN {X 0,Y 184.026,Z 586.061,A -85,B 0,C 180,E1 -27296.176,E2 -27296.176} C_VEL
LIN {X 0,Y 176.905,Z 579.098,A -85,B 0,C 180,E1 -27300.227,E2 -27300.227} C_VEL
LIN {X 0,Y 170.608,Z 570.968,A -85,B 0,C 180,E1 -27304.528,E2 -27304.528} C_VEL
LIN {X 0,Y 165.89,Z 562.9,A -85,B 0,C 180,E1 -27308.396,E2 -27308.396} C_VEL
LIN {X 0,Y 162.13,Z 554.328,A -85,B 0,C 180,E1 -27312.072,E2 -27312.072} C_VEL
LIN {X 0,Y 158.946,Z 545.125,A -85,B 0,C 180,E1 -27315.604,E2 -27315.604} C_VEL
LIN {X 0,Y 156.255,Z 535.477,A -85,B 0,C 180,E1 -27318.871,E2 -27318.871} C_VEL
LIN {X 0,Y 153.866,Z 525.498,A -85,B 0,C 180,E1 -27321.828,E2 -27321.828} C_VEL
LIN {X 0,Y 151.173,Z 513.817,A -85,B 0,C 180,E1 -27324.881,E2 -27324.881} C_VEL
LIN {X 0,Y 147.902,Z 503.295,A -85,B 0,C 180,E1 -27327.798,E2 -27327.798} C_VEL
LIN {X 0,Y 144.807,Z 495.611,A -85,B 0,C 180,E1 -27330.569,E2 -27330.569} C_VEL
LIN {X 0,Y 141.293,Z 487.851,A -85,B 0,C 180,E1 -27334.103,E2 -27334.103} C_VEL
LIN {X 0,Y 137.891,Z 481.192,A -85,B 0,C 180,E1 -27338.119,E2 -27338.119} C_VEL
LIN {X 0,Y 135.727,Z 477.435,A -85,B 0,C 180,E1 -27341.145,E2 -27341.145} C_VEL
LIN {X 0,Y 134.117,Z 474.584,A -85,B 0,C 180,E1 -27343.838,E2 -27343.838} C_VEL
LIN {X 0,Y 131.998,Z 470.783,A -85,B 0,C 180,E1 -27348.437,E2 -27348.437} C_VEL
LIN {X 0,Y 130.151,Z 467.146,A -85,B 0,C 180,E1 -27355.938,E2 -27355.938} C_VEL
LIN {X 0,Y 129.998,Z 466.274,A -85,B 0,C 180,E1 -27358.453,E2 -27358.453} C_VEL
LIN {X 0,Y 129.988,Z 466.212,A -85,B 0,C 180,E1 -27360.776,E2 -27360.776} C_VEL
LIN {X 0,Y 130.153,Z 467.13,A -85,B 0,C 180,E1 -27363.678,E2 -27363.678} C_VEL
LIN {X 0,Y 131.98,Z 470.767,A -85,B 0,C 180,E1 -27371.132,E2 -27371.132} C_VEL
LIN {X 0,Y 134.634,Z 475.456,A -85,B 0,C 180,E1 -27376.686,E2 -27376.686} C_VEL
LIN {X 0,Y 137.036,Z 479.657,A -85,B 0,C 180,E1 -27380.353,E2 -27380.353} C_VEL
LIN {X 0,Y 140.076,Z 485.389,A -85,B 0,C 180,E1 -27384.158,E2 -27384.158} C_VEL
LIN {X 0,Y 142.397,Z 492.19,A -85,B 0,C 180,E1 -27386.893,E2 -27386.893} C_VEL
LIN {X 0,Y 144.457,Z 498.791,A -85,B 0,C 180,E1 -27389.113,E2 -27389.113} C_VEL
LIN {X 0,Y 142.317,Z 519.736,A -85,B 0,C 180,E1 -27389.922,E2 -27389.922} C_VEL
LIN {X 0,Y 139.761,Z 533.214,A -85,B 0,C 180,E1 -27390.733,E2 -27390.733} C_VEL
LIN {X 0,Y 136.387,Z 544.811,A -85,B 0,C 180,E1 -27391.765,E2 -27391.765} C_VEL
LIN {X 0,Y 132.197,Z 555.918,A -85,B 0,C 180,E1 -27393.145,E2 -27393.145} C_VEL
LIN {X 0,Y 128.103,Z 564.913,A -85,B 0,C 180,E1 -27394.624,E2 -27394.624} C_VEL
LIN {X 0,Y 123.462,Z 573.634,A -85,B 0,C 180,E1 -27396.484,E2 -27396.484} C_VEL
LIN {X 0,Y 118.963,Z 581.049,A -85,B 0,C 180,E1 -27398.488,E2 -27398.488} C_VEL
LIN {X 0,Y 112.842,Z 589.839,A -85,B 0,C 180,E1 -27401.638,E2 -27401.638} C_VEL
LIN {X 0,Y 108.232,Z 595.825,A -85,B 0,C 180,E1 -27404.418,E2 -27404.418} C_VEL
LIN {X 0,Y 102.952,Z 602.137,A -85,B 0,C 180,E1 -27408.277,E2 -27408.277} C_VEL
LIN {X 0,Y 98.274,Z 607.413,A -85,B 0,C 180,E1 -27412.566,E2 -27412.566} C_VEL
LIN {X 0,Y 93.204,Z 612.506,A -85,B 0,C 180,E1 -27418.143,E2 -27418.143} C_VEL
LIN {X 0,Y 89.135,Z 616.473,A -85,B 0,C 180,E1 -27424.302,E2 -27424.302} C_VEL
LIN {X 0,Y 86.238,Z 619.416,A -85,B 0,C 180,E1 -27430.977,E2 -27430.977} C_VEL
LIN {X 0,Y 84.953,Z 620.925,A -85,B 0,C 180,E1 -27435.632,E2 -27435.632} C_VEL
LIN {X 0,Y 83.798,Z 622.465,A -85,B 0,C 180,E1 -27445.191,E2 -27445.191} C_VEL
LIN {X 0,Y 83.883,Z 622.753,A -85,B 0,C 180,E1 -27450.001,E2 -27450.001} C_VEL
LIN {X 0,Y 84.13,Z 621.86,A -85,B 0,C 180,E1 -27459.619,E2 -27459.619} C_VEL
LIN {X 0,Y 84.944,Z 620.924,A -85,B 0,C 180,E1 -27464.373,E2 -27464.373} C_VEL
LIN {X 0,Y 88,Z 617.562,A -85,B 0,C 180,E1 -27473.537,E2 -27473.537} C_VEL
LIN {X 0,Y 91.744,Z 613.933,A -85,B 0,C 180,E1 -27479.864,E2 -27479.864} C_VEL
LIN {X 0,Y 94.766,Z 610.989,A -85,B 0,C 180,E1 -27483.795,E2 -27483.795} C_VEL
LIN {X 0,Y 100.092,Z 605.413,A -85,B 0,C 180,E1 -27489.194,E2 -27489.194} C_VEL
LIN {X 0,Y 105.034,Z 599.758,A -85,B 0,C 180,E1 -27493.303,E2 -27493.303} C_VEL
LIN {X 0,Y 110.53,Z 592.956,A -85,B 0,C 180,E1 -27496.99,E2 -27496.99} C_VEL
LIN {X 0,Y 116.483,Z 584.743,A -85,B 0,C 180,E1 -27500.289,E2 -27500.289} C_VEL
LIN {X 0,Y 121.513,Z 576.921,A -85,B 0,C 180,E1 -27502.681,E2 -27502.681} C_VEL
LIN {X 0,Y 126.088,Z 568.843,A -85,B 0,C 180,E1 -27504.606,E2 -27504.606} C_VEL
LIN {X 0,Y 130.825,Z 559.088,A -85,B 0,C 180,E1 -27506.374,E2 -27506.374} C_VEL
LIN {X 0,Y 134.295,Z 550.703,A -85,B 0,C 180,E1 -27507.55,E2 -27507.55} C_VEL
LIN {X 0,Y 137.828,Z 540.202,A -85,B 0,C 180,E1 -27508.661,E2 -27508.661} C_VEL
LIN {X 0,Y 140.527,Z 529.861,A -85,B 0,C 180,E1 -27509.448,E2 -27509.448} C_VEL
LIN {X 0,Y 142.336,Z 519.638,A -85,B 0,C 180,E1 -27510.066,E2 -27510.066} C_VEL
LIN {X 0,Y 144.4,Z 499.941,A -85,B 0,C 180,E1 -27510.813,E2 -27510.813} C_VEL
LIN {X 0,Y 144.386,Z 498.552,A -85,B 0,C 180,E1 -27510.961,E2 -27510.961} C_VEL
LIN {X 0,Y 141.086,Z 488.151,A -85,B 0,C 180,E1 -27514.631,E2 -27514.631} C_VEL
LIN {X 0,Y 139.502,Z 484.259,A -85,B 0,C 180,E1 -27516.51,E2 -27516.51} C_VEL
LIN {X 0,Y 136.357,Z 478.354,A -85,B 0,C 180,E1 -27520.621,E2 -27520.621} C_VEL
LIN {X 0,Y 133.917,Z 474.249,A -85,B 0,C 180,E1 -27524.591,E2 -27524.591} C_VEL
LIN {X 0,Y 131.983,Z 470.736,A -85,B 0,C 180,E1 -27528.869,E2 -27528.869} C_VEL
LIN {X 0,Y 130.06,Z 466.495,A -85,B 0,C 180,E1 -27537.676,E2 -27537.676} C_VEL
LIN {X 0,Y 129.983,Z 466.104,A -85,B 0,C 180,E1 -27539.998,E2 -27539.998} C_VEL
LIN {X 0,Y 130.126,Z 466.894,A -85,B 0,C 180,E1 -27543.675,E2 -27543.675} C_VEL
LIN {X 0,Y 131.717,Z 470.498,A -85,B 0,C 180,E1 -27550.856,E2 -27550.856} C_VEL
LIN {X 0,Y 132.329,Z 471.315,A -85,B 0,C 180,E1 -27552.39,E2 -27552.39} C_VEL
LIN {X 0,Y 134.765,Z 475.718,A -85,B 0,C 180,E1 -27557.301,E2 -27557.301} C_VEL
LIN {X 0,Y 135.181,Z 476.509,A -85,B 0,C 180,E1 -27558.001,E2 -27558.001} C_VEL
LIN {X 0,Y 136.03,Z 478.478,A -85,B 0,C 180,E1 -27559.394,E2 -27559.394} C_VEL
LIN {X 0,Y 136.757,Z 481.012,A -85,B 0,C 180,E1 -27560.627,E2 -27560.627} C_VEL
LIN {X 0,Y 137.982,Z 487.015,A -85,B 0,C 180,E1 -27562.762,E2 -27562.762} C_VEL
LIN {X 0,Y 139.269,Z 493.371,A -85,B 0,C 180,E1 -27564.787,E2 -27564.787} C_VEL
LIN {X 0,Y 140.617,Z 497.644,A -85,B 0,C 180,E1 -27566.449,E2 -27566.449} C_VEL
LIN {X 0,Y 141.195,Z 498.869,A -85,B 0,C 180,E1 -27567.055,E2 -27567.055} C_VEL
LIN {X 0,Y 144.176,Z 506.618,A -85,B 0,C 180,E1 -27570.076,E2 -27570.076} C_VEL
LIN {X 0,Y 146.674,Z 515.192,A -85,B 0,C 180,E1 -27572.719,E2 -27572.719} C_VEL
LIN {X 0,Y 148.797,Z 526.002,A -85,B 0,C 180,E1 -27575.662,E2 -27575.662} C_VEL
LIN {X 0,Y 151.352,Z 538.806,A -85,B 0,C 180,E1 -27579.635,E2 -27579.635} C_VEL
LIN {X 0,Y 154.186,Z 550.699,A -85,B 0,C 180,E1 -27584.034,E2 -27584.034} C_VEL
LIN {X 0,Y 157.106,Z 559.708,A -85,B 0,C 180,E1 -27587.854,E2 -27587.854} C_VEL
LIN {X 0,Y 160.783,Z 568.176,A -85,B 0,C 180,E1 -27591.885,E2 -27591.885} C_VEL
LIN {X 0,Y 165.721,Z 576.344,A -85,B 0,C 180,E1 -27596.251,E2 -27596.251} C_VEL
LIN {X 0,Y 171.737,Z 583.683,A -85,B 0,C 180,E1 -27600.588,E2 -27600.588} C_VEL
LIN {X 0,Y 178.765,Z 590.036,A -85,B 0,C 180,E1 -27604.716,E2 -27604.716} C_VEL
LIN {X 0,Y 188.058,Z 596.135,A -85,B 0,C 180,E1 -27609.11,E2 -27609.11} C_VEL
LIN {X 0,Y 198.396,Z 601.014,A -85,B 0,C 180,E1 -27613.024,E2 -27613.024} C_VEL
LIN {X 0,Y 209.546,Z 604.979,A -85,B 0,C 180,E1 -27616.561,E2 -27616.561} C_VEL
LIN {X 0,Y 221.315,Z 608.236,A -85,B 0,C 180,E1 -27619.867,E2 -27619.867} C_VEL
LIN {X 0,Y 227.39,Z 609.665,A -85,B 0,C 180,E1 -27621.498,E2 -27621.498} C_VEL
LIN {X 0,Y 233.556,Z 610.962,A -85,B 0,C 180,E1 -27623.214,E2 -27623.214} C_VEL
LIN {X 0,Y 239.791,Z 612.248,A -85,B 0,C 180,E1 -27625.192,E2 -27625.192} C_VEL
LIN {X 0,Y 243.485,Z 612.946,A -85,B 0,C 180,E1 -27626.69,E2 -27626.69} C_VEL
LIN {X 0,Y 246.828,Z 613.46,A -85,B 0,C 180,E1 -27628.368,E2 -27628.368} C_VEL
LIN {X 0,Y 248.654,Z 613.617,A -85,B 0,C 180,E1 -27630,E2 -27630} C_VEL
LIN {X 0,Y 246.815,Z 613.46,A -85,B 0,C 180,E1 -27631.631,E2 -27631.631} C_VEL
LIN {X 0,Y 243.477,Z 612.947,A -85,B 0,C 180,E1 -27633.309,E2 -27633.309} C_VEL
LIN {X 0,Y 239.034,Z 612.103,A -85,B 0,C 180,E1 -27635.06,E2 -27635.06} C_VEL
LIN {X 0,Y 233.054,Z 610.863,A -85,B 0,C 180,E1 -27636.928,E2 -27636.928} C_VEL
LIN {X 0,Y 225.685,Z 609.278,A -85,B 0,C 180,E1 -27638.957,E2 -27638.957} C_VEL
LIN {X 0,Y 215.368,Z 606.683,A -85,B 0,C 180,E1 -27641.776,E2 -27641.776} C_VEL
LIN {X 0,Y 200.321,Z 601.809,A -85,B 0,C 180,E1 -27646.299,E2 -27646.299} C_VEL
LIN {X 0,Y 190.899,Z 597.631,A -85,B 0,C 180,E1 -27649.737,E2 -27649.737} C_VEL
LIN {X 0,Y 180.977,Z 591.684,A -85,B 0,C 180,E1 -27654.138,E2 -27654.138} C_VEL
LIN {X 0,Y 174.576,Z 586.441,A -85,B 0,C 180,E1 -27657.67,E2 -27657.67} C_VEL
LIN {X 0,Y 167.93,Z 579.285,A -85,B 0,C 180,E1 -27662.064,E2 -27662.064} C_VEL
LIN {X 0,Y 162.997,Z 572.148,A -85,B 0,C 180,E1 -27666.059,E2 -27666.059} C_VEL
LIN {X 0,Y 158.87,Z 564.081,A -85,B 0,C 180,E1 -27670.13,E2 -27670.13} C_VEL
LIN {X 0,Y 155.36,Z 554.612,A -85,B 0,C 180,E1 -27674.36,E2 -27674.36} C_VEL
LIN {X 0,Y 153.073,Z 546.413,A -85,B 0,C 180,E1 -27677.631,E2 -27677.631} C_VEL
LIN {X 0,Y 150.619,Z 535.61,A -85,B 0,C 180,E1 -27681.414,E2 -27681.414} C_VEL
LIN {X 0,Y 148.621,Z 525.024,A -85,B 0,C 180,E1 -27684.601,E2 -27684.601} C_VEL
LIN {X 0,Y 146.493,Z 514.298,A -85,B 0,C 180,E1 -27687.541,E2 -27687.541} C_VEL
LIN {X 0,Y 143.843,Z 505.657,A -85,B 0,C 180,E1 -27690.251,E2 -27690.251} C_VEL
LIN {X 0,Y 140.633,Z 497.494,A -85,B 0,C 180,E1 -27693.555,E2 -27693.555} C_VEL
LIN {X 0,Y 137.29,Z 490.092,A -85,B 0,C 180,E1 -27697.523,E2 -27697.523} C_VEL
LIN {X 0,Y 134.473,Z 484.517,A -85,B 0,C 180,E1 -27701.574,E2 -27701.574} C_VEL
LIN {X 0,Y 132.542,Z 481.006,A -85,B 0,C 180,E1 -27705.021,E2 -27705.021} C_VEL
LIN {X 0,Y 130.853,Z 477.663,A -85,B 0,C 180,E1 -27709.071,E2 -27709.071} C_VEL
LIN {X 0,Y 129.162,Z 473.52,A -85,B 0,C 180,E1 -27717.663,E2 -27717.663} C_VEL
LIN {X 0,Y 129.121,Z 473.275,A -85,B 0,C 180,E1 -27720.781,E2 -27720.781} C_VEL
LIN {X 0,Y 129.25,Z 474.266,A -85,B 0,C 180,E1 -27723.509,E2 -27723.509} C_VEL
LIN {X 0,Y 131.091,Z 478.146,A -85,B 0,C 180,E1 -27731.208,E2 -27731.208} C_VEL
LIN {X 0,Y 133.214,Z 482.226,A -85,B 0,C 180,E1 -27735.885,E2 -27735.885} C_VEL
LIN {X 0,Y 135.29,Z 486.143,A -85,B 0,C 180,E1 -27739.317,E2 -27739.317} C_VEL
LIN {X 0,Y 137.708,Z 491.02,A -85,B 0,C 180,E1 -27742.634,E2 -27742.634} C_VEL
LIN {X 0,Y 139.681,Z 497.385,A -85,B 0,C 180,E1 -27745.242,E2 -27745.242} C_VEL
LIN {X 0,Y 140.853,Z 501.501,A -85,B 0,C 180,E1 -27746.685,E2 -27746.685} C_VEL
LIN {X 0,Y 138.81,Z 520.266,A -85,B 0,C 180,E1 -27747.415,E2 -27747.415} C_VEL
LIN {X 0,Y 135.733,Z 534.971,A -85,B 0,C 180,E1 -27748.333,E2 -27748.333} C_VEL
LIN {X 0,Y 132.791,Z 544.616,A -85,B 0,C 180,E1 -27749.163,E2 -27749.163} C_VEL
LIN {X 0,Y 128.458,Z 555.723,A -85,B 0,C 180,E1 -27750.496,E2 -27750.496} C_VEL
LIN {X 0,Y 124.203,Z 564.718,A -85,B 0,C 180,E1 -27751.925,E2 -27751.925} C_VEL
LIN {X 0,Y 119.383,Z 573.439,A -85,B 0,C 180,E1 -27753.746,E2 -27753.746} C_VEL
LIN {X 0,Y 114.673,Z 580.854,A -85,B 0,C 180,E1 -27755.706,E2 -27755.706} C_VEL
LIN {X 0,Y 108.247,Z 589.644,A -85,B 0,C 180,E1 -27758.824,E2 -27758.824} C_VEL
LIN {X 0,Y 103.365,Z 595.629,A -85,B 0,C 180,E1 -27761.592,E2 -27761.592} C_VEL
LIN {X 0,Y 97.638,Z 602.049,A -85,B 0,C 180,E1 -27765.575,E2 -27765.575} C_VEL
LIN {X 0,Y 92.706,Z 607.217,A -85,B 0,C 180,E1 -27769.883,E2 -27769.883} C_VEL
LIN {X 0,Y 87.219,Z 612.31,A -85,B 0,C 180,E1 -27775.666,E2 -27775.666} C_VEL
LIN {X 0,Y 82.77,Z 616.277,A -85,B 0,C 180,E1 -27782.162,E2 -27782.162} C_VEL
LIN {X 0,Y 79.521,Z 619.22,A -85,B 0,C 180,E1 -27789.299,E2 -27789.299} C_VEL
LIN {X 0,Y 78.058,Z 620.729,A -85,B 0,C 180,E1 -27794.331,E2 -27794.331} C_VEL
LIN {X 0,Y 76.735,Z 622.27,A -85,B 0,C 180,E1 -27804.747,E2 -27804.747} C_VEL
LIN {X 0,Y 76.781,Z 622.557,A -85,B 0,C 180,E1 -27810.002,E2 -27810.002} C_VEL
LIN {X 0,Y 77.119,Z 621.665,A -85,B 0,C 180,E1 -27820.503,E2 -27820.503} C_VEL
LIN {X 0,Y 78.05,Z 620.728,A -85,B 0,C 180,E1 -27825.674,E2 -27825.674} C_VEL
LIN {X 0,Y 81.507,Z 617.366,A -85,B 0,C 180,E1 -27835.541,E2 -27835.541} C_VEL
LIN {X 0,Y 85.636,Z 613.737,A -85,B 0,C 180,E1 -27842.24,E2 -27842.24} C_VEL
LIN {X 0,Y 88.94,Z 610.793,A -85,B 0,C 180,E1 -27846.346,E2 -27846.346} C_VEL
LIN {X 0,Y 94.688,Z 605.218,A -85,B 0,C 180,E1 -27851.914,E2 -27851.914} C_VEL
LIN {X 0,Y 99.976,Z 599.563,A -85,B 0,C 180,E1 -27856.1,E2 -27856.1} C_VEL
LIN {X 0,Y 105.809,Z 592.76,A -85,B 0,C 180,E1 -27859.805,E2 -27859.805} C_VEL
LIN {X 0,Y 112.071,Z 584.548,A -85,B 0,C 180,E1 -27863.089,E2 -27863.089} C_VEL
LIN {X 0,Y 117.331,Z 576.726,A -85,B 0,C 180,E1 -27865.448,E2 -27865.448} C_VEL
LIN {X 0,Y 122.113,Z 568.648,A -85,B 0,C 180,E1 -27867.322,E2 -27867.322} C_VEL
LIN {X 0,Y 127.031,Z 558.893,A -85,B 0,C 180,E1 -27869.042,E2 -27869.042} C_VEL
LIN {X 0,Y 130.627,Z 550.508,A -85,B 0,C 180,E1 -27870.176,E2 -27870.176} C_VEL
LIN {X 0,Y 134.278,Z 540.007,A -85,B 0,C 180,E1 -27871.245,E2 -27871.245} C_VEL
LIN {X 0,Y 137.152,Z 529.111,A -85,B 0,C 180,E1 -27872.054,E2 -27872.054} C_VEL
LIN {X 0,Y 139.022,Z 518.696,A -85,B 0,C 180,E1 -27872.642,E2 -27872.642} C_VEL
LIN {X 0,Y 140.855,Z 501.485,A -85,B 0,C 180,E1 -27873.315,E2 -27873.315} C_VEL
LIN {X 0,Y 138.233,Z 492.454,A -85,B 0,C 180,E1 -27876.672,E2 -27876.672} C_VEL
LIN {X 0,Y 137.088,Z 489.732,A -85,B 0,C 180,E1 -27878.165,E2 -27878.165} C_VEL
LIN {X 0,Y 134.616,Z 484.718,A -85,B 0,C 180,E1 -27881.743,E2 -27881.743} C_VEL
LIN {X 0,Y 132.45,Z 480.828,A -85,B 0,C 180,E1 -27885.596,E2 -27885.596} C_VEL
LIN {X 0,Y 130.785,Z 477.557,A -85,B 0,C 180,E1 -27889.647,E2 -27889.647} C_VEL
LIN {X 0,Y 129.145,Z 473.418,A -85,B 0,C 180,E1 -27898.439,E2 -27898.439} C_VEL
LIN {X 0,Y 129.118,Z 473.153,A -85,B 0,C 180,E1 -27899.998,E2 -27899.998} C_VEL
LIN {X 0,Y 129.198,Z 473.859,A -85,B 0,C 180,E1 -27903.116,E2 -27903.116} C_VEL
LIN {X 0,Y 131.111,Z 478.157,A -85,B 0,C 180,E1 -27911.642,E2 -27911.642} C_VEL
LIN {X 0,Y 133.313,Z 482.433,A -85,B 0,C 180,E1 -27916.459,E2 -27916.459} C_VEL
LIN {X 0,Y 135.444,Z 486.436,A -85,B 0,C 180,E1 -27919.931,E2 -27919.931} C_VEL
LIN {X 0,Y 138.18,Z 492.021,A -85,B 0,C 180,E1 -27923.609,E2 -27923.609} C_VEL
LIN {X 0,Y 141.195,Z 498.869,A -85,B 0,C 180,E1 -27927.055,E2 -27927.055} C_VEL
LIN {X 0,Y 142.228,Z 501.509,A -85,B 0,C 180,E1 -27928.137,E2 -27928.137} C_VEL
LIN {X 0,Y 142.95,Z 504.703,A -85,B 0,C 180,E1 -27929.002,E2 -27929.002} C_VEL
LIN {X 0,Y 143.54,Z 510.077,A -85,B 0,C 180,E1 -27930.019,E2 -27930.019} C_VEL
LIN {X 0,Y 143.801,Z 519.611,A -85,B 0,C 180,E1 -27931.503,E2 -27931.503} C_VEL
LIN {X 0,Y 143.94,Z 525.04,A -85,B 0,C 180,E1 -27932.634,E2 -27932.634} C_VEL
LIN {X 0,Y 144.156,Z 526.705,A -85,B 0,C 180,E1 -27933.094,E2 -27933.094} C_VEL
LIN {X 0,Y 145.982,Z 539.207,A -85,B 0,C 180,E1 -27937.062,E2 -27937.062} C_VEL
LIN {X 0,Y 147.76,Z 549.299,A -85,B 0,C 180,E1 -27940.842,E2 -27940.842} C_VEL
LIN {X 0,Y 149.873,Z 558.352,A -85,B 0,C 180,E1 -27944.698,E2 -27944.698} C_VEL
LIN {X 0,Y 153.139,Z 568.235,A -85,B 0,C 180,E1 -27949.521,E2 -27949.521} C_VEL
LIN {X 0,Y 156.931,Z 575.801,A -85,B 0,C 180,E1 -27953.715,E2 -27953.715} C_VEL
LIN {X 0,Y 162.769,Z 583.961,A -85,B 0,C 180,E1 -27958.792,E2 -27958.792} C_VEL
LIN {X 0,Y 169.198,Z 590.47,A -85,B 0,C 180,E1 -27963.253,E2 -27963.253} C_VEL
LIN {X 0,Y 175.732,Z 595.34,A -85,B 0,C 180,E1 -27966.898,E2 -27966.898} C_VEL
LIN {X 0,Y 185.465,Z 600.645,A -85,B 0,C 180,E1 -27971.32,E2 -27971.32} C_VEL
LIN {X 0,Y 197.297,Z 605.121,A -85,B 0,C 180,E1 -27975.561,E2 -27975.561} C_VEL
LIN {X 0,Y 207.805,Z 608.095,A -85,B 0,C 180,E1 -27978.744,E2 -27978.744} C_VEL
LIN {X 0,Y 219.966,Z 610.735,A -85,B 0,C 180,E1 -27982.072,E2 -27982.072} C_VEL
LIN {X 0,Y 226.217,Z 611.835,A -85,B 0,C 180,E1 -27983.793,E2 -27983.793} C_VEL
LIN {X 0,Y 232.572,Z 612.829,A -85,B 0,C 180,E1 -27985.707,E2 -27985.707} C_VEL
LIN {X 0,Y 234.94,Z 613.179,A -85,B 0,C 180,E1 -27986.57,E2 -27986.57} C_VEL
LIN {X 0,Y 239.046,Z 613.677,A -85,B 0,C 180,E1 -27988.358,E2 -27988.358} C_VEL
LIN {X 0,Y 241.3,Z 613.819,A -85,B 0,C 180,E1 -27990,E2 -27990} C_VEL
LIN {X 0,Y 238.949,Z 613.672,A -85,B 0,C 180,E1 -27991.685,E2 -27991.685} C_VEL
LIN {X 0,Y 234.938,Z 613.18,A -85,B 0,C 180,E1 -27993.429,E2 -27993.429} C_VEL
LIN {X 0,Y 232.572,Z 612.83,A -85,B 0,C 180,E1 -27994.292,E2 -27994.292} C_VEL
LIN {X 0,Y 226.217,Z 611.836,A -85,B 0,C 180,E1 -27996.205,E2 -27996.205} C_VEL
LIN {X 0,Y 219.965,Z 610.736,A -85,B 0,C 180,E1 -27997.926,E2 -27997.926} C_VEL
LIN {X 0,Y 205.843,Z 607.613,A -85,B 0,C 180,E1 -28001.82,E2 -28001.82} C_VEL
LIN {X 0,Y 190.738,Z 602.83,A -85,B 0,C 180,E1 -28006.669,E2 -28006.669} C_VEL
LIN {X 0,Y 180.463,Z 598.107,A -85,B 0,C 180,E1 -28010.831,E2 -28010.831} C_VEL
LIN {X 0,Y 171.282,Z 592.19,A -85,B 0,C 180,E1 -28015.488,E2 -28015.488} C_VEL
LIN {X 0,Y 164.343,Z 585.776,A -85,B 0,C 180,E1 -28020.009,E2 -28020.009} C_VEL
LIN {X 0,Y 159.202,Z 579.363,A -85,B 0,C 180,E1 -28024.138,E2 -28024.138} C_VEL
LIN {X 0,Y 154.844,Z 571.943,A -85,B 0,C 180,E1 -28028.472,E2 -28028.472} C_VEL
LIN {X 0,Y 151.841,Z 564.86,A -85,B 0,C 180,E1 -28032.223,E2 -28032.223} C_VEL
LIN {X 0,Y 148.912,Z 554.985,A -85,B 0,C 180,E1 -28036.801,E2 -28036.801} C_VEL
LIN {X 0,Y 147.038,Z 545.711,A -85,B 0,C 180,E1 -28040.542,E2 -28040.542} C_VEL
LIN {X 0,Y 145.59,Z 536.865,A -85,B 0,C 180,E1 -28043.724,E2 -28043.724} C_VEL
LIN {X 0,Y 144.028,Z 525.856,A -85,B 0,C 180,E1 -28047.145,E2 -28047.145} C_VEL
LIN {X 0,Y 142.299,Z 515.913,A -85,B 0,C 180,E1 -28050.1,E2 -28050.1} C_VEL
LIN {X 0,Y 140.041,Z 508.114,A -85,B 0,C 180,E1 -28052.849,E2 -28052.849} C_VEL
LIN {X 0,Y 136.875,Z 499.947,A -85,B 0,C 180,E1 -28056.628,E2 -28056.628} C_VEL
LIN {X 0,Y 134.17,Z 493.748,A -85,B 0,C 180,E1 -28060.452,E2 -28060.452} C_VEL
LIN {X 0,Y 132.058,Z 489.484,A -85,B 0,C 180,E1 -28064.075,E2 -28064.075} C_VEL
LIN {X 0,Y 130.939,Z 487.291,A -85,B 0,C 180,E1 -28066.419,E2 -28066.419} C_VEL
LIN {X 0,Y 129.697,Z 484.473,A -85,B 0,C 180,E1 -28069.808,E2 -28069.808} C_VEL
LIN {X 0,Y 128.261,Z 480.426,A -85,B 0,C 180,E1 -28078.432,E2 -28078.432} C_VEL
LIN {X 0,Y 128.255,Z 480.321,A -85,B 0,C 180,E1 -28080.787,E2 -28080.787} C_VEL
LIN {X 0,Y 129.88,Z 484.883,A -85,B 0,C 180,E1 -28090.377,E2 -28090.377} C_VEL
LIN {X 0,Y 131.729,Z 488.789,A -85,B 0,C 180,E1 -28094.879,E2 -28094.879} C_VEL
LIN {X 0,Y 133.511,Z 492.414,A -85,B 0,C 180,E1 -28098.116,E2 -28098.116} C_VEL
LIN {X 0,Y 135.589,Z 497.061,A -85,B 0,C 180,E1 -28101.276,E2 -28101.276} C_VEL
LIN {X 0,Y 137.518,Z 504.182,A -85,B 0,C 180,E1 -28104.134,E2 -28104.134} C_VEL
LIN {X 0,Y 135.55,Z 520.987,A -85,B 0,C 180,E1 -28104.789,E2 -28104.789} C_VEL
LIN {X 0,Y 132.512,Z 534.776,A -85,B 0,C 180,E1 -28105.631,E2 -28105.631} C_VEL
LIN {X 0,Y 129.486,Z 544.421,A -85,B 0,C 180,E1 -28106.423,E2 -28106.423} C_VEL
LIN {X 0,Y 125.012,Z 555.528,A -85,B 0,C 180,E1 -28107.697,E2 -28107.697} C_VEL
LIN {X 0,Y 120.596,Z 564.523,A -85,B 0,C 180,E1 -28109.058,E2 -28109.058} C_VEL
LIN {X 0,Y 115.588,Z 573.244,A -85,B 0,C 180,E1 -28110.818,E2 -28110.818} C_VEL
LIN {X 0,Y 110.676,Z 580.659,A -85,B 0,C 180,E1 -28112.717,E2 -28112.717} C_VEL
LIN {X 0,Y 103.934,Z 589.448,A -85,B 0,C 180,E1 -28115.766,E2 -28115.766} C_VEL
LIN {X 0,Y 98.788,Z 595.434,A -85,B 0,C 180,E1 -28118.507,E2 -28118.507} C_VEL
LIN {X 0,Y 92.8,Z 601.744,A -85,B 0,C 180,E1 -28122.408,E2 -28122.408} C_VEL
LIN {X 0,Y 87.302,Z 607.076,A -85,B 0,C 180,E1 -28126.921,E2 -28126.921} C_VEL
LIN {X 0,Y 81.424,Z 612.114,A -85,B 0,C 180,E1 -28132.832,E2 -28132.832} C_VEL
LIN {X 0,Y 76.544,Z 616.082,A -85,B 0,C 180,E1 -28139.671,E2 -28139.671} C_VEL
LIN {X 0,Y 72.893,Z 619.024,A -85,B 0,C 180,E1 -28147.317,E2 -28147.317} C_VEL
LIN {X 0,Y 71.221,Z 620.533,A -85,B 0,C 180,E1 -28152.782,E2 -28152.782} C_VEL
LIN {X 0,Y 69.647,Z 622.075,A -85,B 0,C 180,E1 -28164.21,E2 -28164.21} C_VEL
LIN {X 0,Y 69.678,Z 622.362,A -85,B 0,C 180,E1 -28170.002,E2 -28170.002} C_VEL
LIN {X 0,Y 70.14,Z 621.469,A -85,B 0,C 180,E1 -28181.562,E2 -28181.562} C_VEL
LIN {X 0,Y 71.215,Z 620.532,A -85,B 0,C 180,E1 -28187.223,E2 -28187.223} C_VEL
LIN {X 0,Y 75.135,Z 617.17,A -85,B 0,C 180,E1 -28197.886,E2 -28197.886} C_VEL
LIN {X 0,Y 79.698,Z 613.541,A -85,B 0,C 180,E1 -28204.974,E2 -28204.974} C_VEL
LIN {X 0,Y 85.336,Z 608.81,A -85,B 0,C 180,E1 -28211.214,E2 -28211.214} C_VEL
LIN {X 0,Y 91.694,Z 602.838,A -85,B 0,C 180,E1 -28216.728,E2 -28216.728} C_VEL
LIN {X 0,Y 97.577,Z 596.743,A -85,B 0,C 180,E1 -28220.74,E2 -28220.74} C_VEL
LIN {X 0,Y 102.65,Z 591.005,A -85,B 0,C 180,E1 -28223.561,E2 -28223.561} C_VEL
LIN {X 0,Y 107.953,Z 584.353,A -85,B 0,C 180,E1 -28226.105,E2 -28226.105} C_VEL
LIN {X 0,Y 113.453,Z 576.531,A -85,B 0,C 180,E1 -28228.404,E2 -28228.404} C_VEL
LIN {X 0,Y 118.434,Z 568.453,A -85,B 0,C 180,E1 -28230.212,E2 -28230.212} C_VEL
LIN {X 0,Y 123.53,Z 558.698,A -85,B 0,C 180,E1 -28231.866,E2 -28231.866} C_VEL
LIN {X 0,Y 127.247,Z 550.313,A -85,B 0,C 180,E1 -28232.95,E2 -28232.95} C_VEL
LIN {X 0,Y 131.013,Z 539.813,A -85,B 0,C 180,E1 -28233.966,E2 -28233.966} C_VEL
LIN {X 0,Y 133.882,Z 529.324,A -85,B 0,C 180,E1 -28234.714,E2 -28234.714} C_VEL
LIN {X 0,Y 135.802,Z 519.248,A -85,B 0,C 180,E1 -28235.271,E2 -28235.271} C_VEL
LIN {X 0,Y 137.518,Z 504.177,A -85,B 0,C 180,E1 -28235.866,E2 -28235.866} C_VEL
LIN {X 0,Y 135.654,Z 497.207,A -85,B 0,C 180,E1 -28238.634,E2 -28238.634} C_VEL
LIN {X 0,Y 133.514,Z 492.388,A -85,B 0,C 180,E1 -28241.885,E2 -28241.885} C_VEL
LIN {X 0,Y 131.137,Z 487.547,A -85,B 0,C 180,E1 -28246.389,E2 -28246.389} C_VEL
LIN {X 0,Y 129.679,Z 484.445,A -85,B 0,C 180,E1 -28250.248,E2 -28250.248} C_VEL
LIN {X 0,Y 128.277,Z 480.486,A -85,B 0,C 180,E1 -28258.428,E2 -28258.428} C_VEL
LIN {X 0,Y 128.246,Z 480.302,A -85,B 0,C 180,E1 -28260.783,E2 -28260.783} C_VEL
LIN {X 0,Y 128.298,Z 481.023,A -85,B 0,C 180,E1 -28262.942,E2 -28262.942} C_VEL
LIN {X 0,Y 129.907,Z 484.939,A -85,B 0,C 180,E1 -28270.842,E2 -28270.842} C_VEL
LIN {X 0,Y 131.869,Z 489.097,A -85,B 0,C 180,E1 -28275.552,E2 -28275.552} C_VEL
LIN {X 0,Y 133.621,Z 492.643,A -85,B 0,C 180,E1 -28278.682,E2 -28278.682} C_VEL
LIN {X 0,Y 136.279,Z 498.512,A -85,B 0,C 180,E1 -28282.585,E2 -28282.585} C_VEL
LIN {X 0,Y 139.277,Z 506.135,A -85,B 0,C 180,E1 -28286.3,E2 -28286.3} C_VEL
LIN {X 0,Y 141.583,Z 513.22,A -85,B 0,C 180,E1 -28289.045,E2 -28289.045} C_VEL
LIN {X 0,Y 143.477,Z 522.065,A -85,B 0,C 180,E1 -28291.772,E2 -28291.772} C_VEL
LIN {X 0,Y 144.156,Z 526.705,A -85,B 0,C 180,E1 -28293.094,E2 -28293.094} C_VEL
LIN {X 0,Y 144.528,Z 531.655,A -85,B 0,C 180,E1 -28294.366,E2 -28294.366} C_VEL
LIN {X 0,Y 143.704,Z 540.421,A -85,B 0,C 180,E1 -28296.177,E2 -28296.177} C_VEL
LIN {X 0,Y 142.665,Z 548.851,A -85,B 0,C 180,E1 -28298.179,E2 -28298.179} C_VEL
LIN {X 0,Y 142.611,Z 553.275,A -85,B 0,C 180,E1 -28299.738,E2 -28299.738} C_VEL
LIN {X 0,Y 143.957,Z 560.701,A -85,B 0,C 180,E1 -28303.114,E2 -28303.114} C_VEL
LIN {X 0,Y 146.457,Z 569.727,A -85,B 0,C 180,E1 -28307.792,E2 -28307.792} C_VEL
LIN {X 0,Y 149.348,Z 576.685,A -85,B 0,C 180,E1 -28311.846,E2 -28311.846} C_VEL
LIN {X 0,Y 154.008,Z 584.239,A -85,B 0,C 180,E1 -28316.797,E2 -28316.797} C_VEL
LIN {X 0,Y 159.822,Z 590.809,A -85,B 0,C 180,E1 -28321.576,E2 -28321.576} C_VEL
LIN {X 0,Y 165.947,Z 595.828,A -85,B 0,C 180,E1 -28325.574,E2 -28325.574} C_VEL
LIN {X 0,Y 175.296,Z 601.25,A -85,B 0,C 180,E1 -28330.414,E2 -28330.414} C_VEL
LIN {X 0,Y 185.712,Z 605.443,A -85,B 0,C 180,E1 -28334.638,E2 -28334.638} C_VEL
LIN {X 0,Y 194.342,Z 608,A -85,B 0,C 180,E1 -28337.521,E2 -28337.521} C_VEL
LIN {X 0,Y 206.327,Z 610.648,A -85,B 0,C 180,E1 -28341.036,E2 -28341.036} C_VEL
LIN {X 0,Y 219.093,Z 612.656,A -85,B 0,C 180,E1 -28344.477,E2 -28344.477} C_VEL
LIN {X 0,Y 225.828,Z 613.428,A -85,B 0,C 180,E1 -28346.431,E2 -28346.431} C_VEL
LIN {X 0,Y 231.968,Z 613.955,A -85,B 0,C 180,E1 -28348.823,E2 -28348.823} C_VEL
LIN {X 0,Y 233.822,Z 614.025,A -85,B 0,C 180,E1 -28349.999,E2 -28349.999} C_VEL
LIN {X 0,Y 231.968,Z 613.955,A -85,B 0,C 180,E1 -28351.175,E2 -28351.175} C_VEL
LIN {X 0,Y 225.826,Z 613.429,A -85,B 0,C 180,E1 -28353.568,E2 -28353.568} C_VEL
LIN {X 0,Y 218.899,Z 612.632,A -85,B 0,C 180,E1 -28355.574,E2 -28355.574} C_VEL
LIN {X 0,Y 206.327,Z 610.648,A -85,B 0,C 180,E1 -28358.963,E2 -28358.963} C_VEL
LIN {X 0,Y 194.028,Z 607.946,A -85,B 0,C 180,E1 -28362.551,E2 -28362.551} C_VEL
LIN {X 0,Y 180.418,Z 603.521,A -85,B 0,C 180,E1 -28367.383,E2 -28367.383} C_VEL
LIN {X 0,Y 170.855,Z 598.946,A -85,B 0,C 180,E1 -28371.727,E2 -28371.727} C_VEL
LIN {X 0,Y 163.831,Z 594.28,A -85,B 0,C 180,E1 -28375.733,E2 -28375.733} C_VEL
LIN {X 0,Y 156.234,Z 586.966,A -85,B 0,C 180,E1 -28381.277,E2 -28381.277} C_VEL
LIN {X 0,Y 150.786,Z 579.308,A -85,B 0,C 180,E1 -28386.488,E2 -28386.488} C_VEL
LIN {X 0,Y 147.681,Z 572.926,A -85,B 0,C 180,E1 -28390.413,E2 -28390.413} C_VEL
LIN {X 0,Y 144.791,Z 563.923,A -85,B 0,C 180,E1 -28395.269,E2 -28395.269} C_VEL
LIN {X 0,Y 142.914,Z 555.283,A -85,B 0,C 180,E1 -28399.409,E2 -28399.409} C_VEL
LIN {X 0,Y 141.546,Z 545.616,A -85,B 0,C 180,E1 -28403.431,E2 -28403.431} C_VEL
LIN {X 0,Y 140.665,Z 536.684,A -85,B 0,C 180,E1 -28406.663,E2 -28406.663} C_VEL
LIN {X 0,Y 139.596,Z 525.574,A -85,B 0,C 180,E1 -28410.19,E2 -28410.19} C_VEL
LIN {X 0,Y 138.204,Z 516.925,A -85,B 0,C 180,E1 -28413.072,E2 -28413.072} C_VEL
LIN {X 0,Y 136.091,Z 509.698,A -85,B 0,C 180,E1 -28416.107,E2 -28416.107} C_VEL
LIN {X 0,Y 133.783,Z 503.473,A -85,B 0,C 180,E1 -28419.408,E2 -28419.408} C_VEL
LIN {X 0,Y 131.733,Z 498.552,A -85,B 0,C 180,E1 -28422.839,E2 -28422.839} C_VEL
LIN {X 0,Y 129.77,Z 494.223,A -85,B 0,C 180,E1 -28426.976,E2 -28426.976} C_VEL
LIN {X 0,Y 128.464,Z 491.22,A -85,B 0,C 180,E1 -28430.853,E2 -28430.853} C_VEL
LIN {X 0,Y 127.391,Z 487.511,A -85,B 0,C 180,E1 -28438.421,E2 -28438.421} C_VEL
LIN {X 0,Y 127.384,Z 487.36,A -85,B 0,C 180,E1 -28440.595,E2 -28440.595} C_VEL
LIN {X 0,Y 128.718,Z 491.761,A -85,B 0,C 180,E1 -28449.628,E2 -28449.628} C_VEL
LIN {X 0,Y 130.335,Z 495.455,A -85,B 0,C 180,E1 -28453.961,E2 -28453.961} C_VEL
LIN {X 0,Y 132.022,Z 499.203,A -85,B 0,C 180,E1 -28457.297,E2 -28457.297} C_VEL
LIN {X 0,Y 133.513,Z 502.941,A -85,B 0,C 180,E1 -28459.809,E2 -28459.809} C_VEL
LIN {X 0,Y 134.451,Z 507.016,A -85,B 0,C 180,E1 -28461.465,E2 -28461.465} C_VEL
LIN {X 0,Y 132.556,Z 521.976,A -85,B 0,C 180,E1 -28462.065,E2 -28462.065} C_VEL
LIN {X 0,Y 129.593,Z 534.581,A -85,B 0,C 180,E1 -28462.794,E2 -28462.794} C_VEL
LIN {X 0,Y 126.451,Z 544.328,A -85,B 0,C 180,E1 -28463.557,E2 -28463.557} C_VEL
LIN {X 0,Y 121.875,Z 555.333,A -85,B 0,C 180,E1 -28464.742,E2 -28464.742} C_VEL
LIN {X 0,Y 117.311,Z 564.328,A -85,B 0,C 180,E1 -28466.024,E2 -28466.024} C_VEL
LIN {X 0,Y 112.105,Z 573.049,A -85,B 0,C 180,E1 -28467.689,E2 -28467.689} C_VEL
LIN {X 0,Y 107.004,Z 580.464,A -85,B 0,C 180,E1 -28469.515,E2 -28469.515} C_VEL
LIN {X 0,Y 99.936,Z 589.252,A -85,B 0,C 180,E1 -28472.449,E2 -28472.449} C_VEL
LIN {X 0,Y 94.527,Z 595.239,A -85,B 0,C 180,E1 -28475.134,E2 -28475.134} C_VEL
LIN {X 0,Y 88.147,Z 601.548,A -85,B 0,C 180,E1 -28478.982,E2 -28478.982} C_VEL
LIN {X 0,Y 81.436,Z 607.524,A -85,B 0,C 180,E1 -28484.219,E2 -28484.219} C_VEL
LIN {X 0,Y 75.866,Z 611.918,A -85,B 0,C 180,E1 -28489.577,E2 -28489.577} C_VEL
LIN {X 0,Y 70.491,Z 615.886,A -85,B 0,C 180,E1 -28496.748,E2 -28496.748} C_VEL
LIN {X 0,Y 66.354,Z 618.828,A -85,B 0,C 180,E1 -28504.936,E2 -28504.936} C_VEL
LIN {X 0,Y 64.456,Z 620.337,A -85,B 0,C 180,E1 -28510.909,E2 -28510.909} C_VEL
LIN {X 0,Y 62.577,Z 621.88,A -85,B 0,C 180,E1 -28523.554,E2 -28523.554} C_VEL
LIN {X 0,Y 62.569,Z 622.167,A -85,B 0,C 180,E1 -28530.002,E2 -28530.002} C_VEL
LIN {X 0,Y 63.177,Z 621.274,A -85,B 0,C 180,E1 -28542.857,E2 -28542.857} C_VEL
LIN {X 0,Y 64.45,Z 620.336,A -85,B 0,C 180,E1 -28549.097,E2 -28549.097} C_VEL
LIN {X 0,Y 68.918,Z 616.974,A -85,B 0,C 180,E1 -28560.658,E2 -28560.658} C_VEL
LIN {X 0,Y 73.973,Z 613.345,A -85,B 0,C 180,E1 -28568.139,E2 -28568.139} C_VEL
LIN {X 0,Y 80.104,Z 608.614,A -85,B 0,C 180,E1 -28574.58,E2 -28574.58} C_VEL
LIN {X 0,Y 85.783,Z 603.733,A -85,B 0,C 180,E1 -28579.275,E2 -28579.275} C_VEL
LIN {X 0,Y 91.935,Z 597.859,A -85,B 0,C 180,E1 -28583.388,E2 -28583.388} C_VEL
LIN {X 0,Y 97.243,Z 592.37,A -85,B 0,C 180,E1 -28586.217,E2 -28586.217} C_VEL
LIN {X 0,Y 104.161,Z 584.158,A -85,B 0,C 180,E1 -28589.348,E2 -28589.348} C_VEL
LIN {X 0,Y 109.9,Z 576.336,A -85,B 0,C 180,E1 -28591.559,E2 -28591.559} C_VEL
LIN {X 0,Y 115.075,Z 568.258,A -85,B 0,C 180,E1 -28593.278,E2 -28593.278} C_VEL
LIN {X 0,Y 120.339,Z 558.503,A -85,B 0,C 180,E1 -28594.855,E2 -28594.855} C_VEL
LIN {X 0,Y 124.17,Z 550.144,A -85,B 0,C 180,E1 -28595.865,E2 -28595.865} C_VEL
LIN {X 0,Y 127.996,Z 539.812,A -85,B 0,C 180,E1 -28596.807,E2 -28596.807} C_VEL
LIN {X 0,Y 130.991,Z 529.178,A -85,B 0,C 180,E1 -28597.525,E2 -28597.525} C_VEL
LIN {X 0,Y 133.081,Z 518.399,A -85,B 0,C 180,E1 -28598.077,E2 -28598.077} C_VEL
LIN {X 0,Y 134.454,Z 506.986,A -85,B 0,C 180,E1 -28598.536,E2 -28598.536} C_VEL
LIN {X 0,Y 133.274,Z 502.112,A -85,B 0,C 180,E1 -28600.605,E2 -28600.605} C_VEL
LIN {X 0,Y 131.095,Z 497.093,A -85,B 0,C 180,E1 -28604.45,E2 -28604.45} C_VEL
LIN {X 0,Y 129.647,Z 493.94,A -85,B 0,C 180,E1 -28607.674,E2 -28607.674} C_VEL
LIN {X 0,Y 128.437,Z 491.146,A -85,B 0,C 180,E1 -28611.344,E2 -28611.344} C_VEL
LIN {X 0,Y 127.384,Z 487.42,A -85,B 0,C 180,E1 -28619.208,E2 -28619.208} C_VEL
LIN {X 0,Y 127.39,Z 487.522,A -85,B 0,C 180,E1 -28621.579,E2 -28621.579} C_VEL
LIN {X 0,Y 128.726,Z 491.716,A -85,B 0,C 180,E1 -28630.021,E2 -28630.021} C_VEL
LIN {X 0,Y 130.354,Z 495.492,A -85,B 0,C 180,E1 -28634.388,E2 -28634.388} C_VEL
LIN {X 0,Y 131.974,Z 499.11,A -85,B 0,C 180,E1 -28637.601,E2 -28637.601} C_VEL
LIN {X 0,Y 134.192,Z 504.477,A -85,B 0,C 180,E1 -28641.203,E2 -28641.203} C_VEL
LIN {X 0,Y 136.687,Z 511.658,A -85,B 0,C 180,E1 -28644.793,E2 -28644.793} C_VEL
LIN {X 0,Y 138.605,Z 518.686,A -85,B 0,C 180,E1 -28647.559,E2 -28647.559} C_VEL
LIN {X 0,Y 139.838,Z 527.783,A -85,B 0,C 180,E1 -28650.451,E2 -28650.451} C_VEL
LIN {X 0,Y 141.09,Z 540.894,A -85,B 0,C 180,E1 -28654.812,E2 -28654.812} C_VEL
LIN {X 0,Y 142.114,Z 549.664,A -85,B 0,C 180,E1 -28658.178,E2 -28658.178} C_VEL
LIN {X 0,Y 142.611,Z 553.275,A -85,B 0,C 180,E1 -28659.738,E2 -28659.738} C_VEL
LIN {X 0,Y 142.894,Z 557.557,A -85,B 0,C 180,E1 -28661.374,E2 -28661.374} C_VEL
LIN {X 0,Y 141.826,Z 565.131,A -85,B 0,C 180,E1 -28663.945,E2 -28663.945} C_VEL
LIN {X 0,Y 140.942,Z 572.211,A -85,B 0,C 180,E1 -28666.704,E2 -28666.704} C_VEL
LIN {X 0,Y 141.373,Z 575.718,A -85,B 0,C 180,E1 -28668.605,E2 -28668.605} C_VEL
LIN {X 0,Y 144.629,Z 582.828,A -85,B 0,C 180,E1 -28673.353,E2 -28673.353} C_VEL
LIN {X 0,Y 149.975,Z 590.214,A -85,B 0,C 180,E1 -28678.97,E2 -28678.97} C_VEL
LIN {X 0,Y 156.323,Z 596.238,A -85,B 0,C 180,E1 -28684.045,E2 -28684.045} C_VEL
LIN {X 0,Y 165.202,Z 601.82,A -85,B 0,C 180,E1 -28689.373,E2 -28689.373} C_VEL
LIN {X 0,Y 175.435,Z 606.103,A -85,B 0,C 180,E1 -28694.034,E2 -28694.034} C_VEL
LIN {X 0,Y 186.747,Z 609.309,A -85,B 0,C 180,E1 -28698.085,E2 -28698.085} C_VEL
LIN {X 0,Y 199.548,Z 611.782,A -85,B 0,C 180,E1 -28701.901,E2 -28701.901} C_VEL
LIN {X 0,Y 211.595,Z 613.334,A -85,B 0,C 180,E1 -28705.145,E2 -28705.145} C_VEL
LIN {X 0,Y 218.168,Z 613.931,A -85,B 0,C 180,E1 -28706.972,E2 -28706.972} C_VEL
LIN {X 0,Y 221.905,Z 614.131,A -85,B 0,C 180,E1 -28708.185,E2 -28708.185} C_VEL
LIN {X 0,Y 224.908,Z 614.212,A -85,B 0,C 180,E1 -28709.31,E2 -28709.31} C_VEL
LIN {X 0,Y 226.181,Z 614.235,A -85,B 0,C 180,E1 -28709.999,E2 -28709.999} C_VEL
LIN {X 0,Y 224.908,Z 614.212,A -85,B 0,C 180,E1 -28710.688,E2 -28710.688} C_VEL
LIN {X 0,Y 221.903,Z 614.131,A -85,B 0,C 180,E1 -28711.814,E2 -28711.814} C_VEL
LIN {X 0,Y 218.168,Z 613.932,A -85,B 0,C 180,E1 -28713.026,E2 -28713.026} C_VEL
LIN {X 0,Y 207.987,Z 612.966,A -85,B 0,C 180,E1 -28715.818,E2 -28715.818} C_VEL
LIN {X 0,Y 192.709,Z 610.63,A -85,B 0,C 180,E1 -28720.05,E2 -28720.05} C_VEL
LIN {X 0,Y 180.969,Z 607.87,A -85,B 0,C 180,E1 -28723.866,E2 -28723.866} C_VEL
LIN {X 0,Y 170.187,Z 604.123,A -85,B 0,C 180,E1 -28728.236,E2 -28728.236} C_VEL
LIN {X 0,Y 160.58,Z 599.222,A -85,B 0,C 180,E1 -28733.21,E2 -28733.21} C_VEL
LIN {X 0,Y 153.843,Z 594.152,A -85,B 0,C 180,E1 -28737.794,E2 -28737.794} C_VEL
LIN {X 0,Y 147.412,Z 587.111,A -85,B 0,C 180,E1 -28743.457,E2 -28743.457} C_VEL
LIN {X 0,Y 143.318,Z 580.393,A -85,B 0,C 180,E1 -28748.319,E2 -28748.319} C_VEL
LIN {X 0,Y 140.246,Z 572.439,A -85,B 0,C 180,E1 -28753.401,E2 -28753.401} C_VEL
LIN {X 0,Y 138.54,Z 564.838,A -85,B 0,C 180,E1 -28757.662,E2 -28757.662} C_VEL
LIN {X 0,Y 137.334,Z 555.763,A -85,B 0,C 180,E1 -28762.116,E2 -28762.116} C_VEL
LIN {X 0,Y 136.62,Z 546.635,A -85,B 0,C 180,E1 -28766.046,E2 -28766.046} C_VEL
LIN {X 0,Y 136.165,Z 536.491,A -85,B 0,C 180,E1 -28769.789,E2 -28769.789} C_VEL
LIN {X 0,Y 135.596,Z 526.427,A -85,B 0,C 180,E1 -28773.136,E2 -28773.136} C_VEL
LIN {X 0,Y 134.734,Z 519.983,A -85,B 0,C 180,E1 -28775.543,E2 -28775.543} C_VEL
LIN {X 0,Y 132.858,Z 512.675,A -85,B 0,C 180,E1 -28778.98,E2 -28778.98} C_VEL
LIN {X 0,Y 130.887,Z 506.873,A -85,B 0,C 180,E1 -28782.523,E2 -28782.523} C_VEL
LIN {X 0,Y 129.286,Z 502.89,A -85,B 0,C 180,E1 -28785.843,E2 -28785.843} C_VEL
LIN {X 0,Y 128.244,Z 500.381,A -85,B 0,C 180,E1 -28788.542,E2 -28788.542} C_VEL
LIN {X 0,Y 127.345,Z 498.019,A -85,B 0,C 180,E1 -28791.672,E2 -28791.672} C_VEL
LIN {X 0,Y 126.51,Z 494.426,A -85,B 0,C 180,E1 -28799.286,E2 -28799.286} C_VEL
LIN {X 0,Y 126.51,Z 494.513,A -85,B 0,C 180,E1 -28800.718,E2 -28800.718} C_VEL
LIN {X 0,Y 127.597,Z 498.633,A -85,B 0,C 180,E1 -28808.913,E2 -28808.913} C_VEL
LIN {X 0,Y 129.014,Z 502.202,A -85,B 0,C 180,E1 -28813.114,E2 -28813.114} C_VEL
LIN {X 0,Y 130.593,Z 506.032,A -85,B 0,C 180,E1 -28816.514,E2 -28816.514} C_VEL
LIN {X 0,Y 131.467,Z 508.746,A -85,B 0,C 180,E1 -28818.206,E2 -28818.206} C_VEL
LIN {X 0,Y 131.687,Z 509.87,A -85,B 0,C 180,E1 -28818.678,E2 -28818.678} C_VEL
LIN {X 0,Y 129.645,Z 523.683,A -85,B 0,C 180,E1 -28819.255,E2 -28819.255} C_VEL
LIN {X 0,Y 126.579,Z 535.772,A -85,B 0,C 180,E1 -28819.941,E2 -28819.941} C_VEL
LIN {X 0,Y 123.608,Z 544.572,A -85,B 0,C 180,E1 -28820.583,E2 -28820.583} C_VEL
LIN {X 0,Y 119.081,Z 555.138,A -85,B 0,C 180,E1 -28821.641,E2 -28821.641} C_VEL
LIN {X 0,Y 114.37,Z 564.132,A -85,B 0,C 180,E1 -28822.822,E2 -28822.822} C_VEL
LIN {X 0,Y 108.984,Z 572.853,A -85,B 0,C 180,E1 -28824.378,E2 -28824.378} C_VEL
LIN {X 0,Y 103.688,Z 580.269,A -85,B 0,C 180,E1 -28826.096,E2 -28826.096} C_VEL
LIN {X 0,Y 96.303,Z 589.057,A -85,B 0,C 180,E1 -28828.872,E2 -28828.872} C_VEL
LIN {X 0,Y 90.612,Z 595.043,A -85,B 0,C 180,E1 -28831.445,E2 -28831.445} C_VEL
LIN {X 0,Y 83.832,Z 601.352,A -85,B 0,C 180,E1 -28835.18,E2 -28835.18} C_VEL
LIN {X 0,Y 77.421,Z 606.704,A -85,B 0,C 180,E1 -28839.68,E2 -28839.68} C_VEL
LIN {X 0,Y 70.596,Z 611.722,A -85,B 0,C 180,E1 -28845.827,E2 -28845.827} C_VEL
LIN {X 0,Y 64.659,Z 615.691,A -85,B 0,C 180,E1 -28853.29,E2 -28853.29} C_VEL
LIN {X 0,Y 59.957,Z 618.632,A -85,B 0,C 180,E1 -28862.042,E2 -28862.042} C_VEL
LIN {X 0,Y 57.765,Z 620.141,A -85,B 0,C 180,E1 -28868.595,E2 -28868.595} C_VEL
LIN {X 0,Y 55.531,Z 621.685,A -85,B 0,C 180,E1 -28882.731,E2 -28882.731} C_VEL
LIN {X 0,Y 55.48,Z 621.972,A -85,B 0,C 180,E1 -28890.002,E2 -28890.002} C_VEL
LIN {X 0,Y 56.266,Z 621.078,A -85,B 0,C 180,E1 -28904.469,E2 -28904.469} C_VEL
LIN {X 0,Y 57.76,Z 620.141,A -85,B 0,C 180,E1 -28911.411,E2 -28911.411} C_VEL
LIN {X 0,Y 62.9,Z 616.779,A -85,B 0,C 180,E1 -28923.965,E2 -28923.965} C_VEL
LIN {X 0,Y 68.501,Z 613.149,A -85,B 0,C 180,E1 -28931.828,E2 -28931.828} C_VEL
LIN {X 0,Y 75.188,Z 608.418,A -85,B 0,C 180,E1 -28938.4,E2 -28938.4} C_VEL
LIN {X 0,Y 81.287,Z 603.536,A -85,B 0,C 180,E1 -28943.107,E2 -28943.107} C_VEL
LIN {X 0,Y 87.87,Z 597.663,A -85,B 0,C 180,E1 -28947.121,E2 -28947.121} C_VEL
LIN {X 0,Y 93.46,Z 592.174,A -85,B 0,C 180,E1 -28949.858,E2 -28949.858} C_VEL
LIN {X 0,Y 100.724,Z 583.963,A -85,B 0,C 180,E1 -28952.828,E2 -28952.828} C_VEL
LIN {X 0,Y 106.705,Z 576.141,A -85,B 0,C 180,E1 -28954.91,E2 -28954.91} C_VEL
LIN {X 0,Y 112.063,Z 568.063,A -85,B 0,C 180,E1 -28956.521,E2 -28956.521} C_VEL
LIN {X 0,Y 117.504,Z 558.308,A -85,B 0,C 180,E1 -28957.983,E2 -28957.983} C_VEL
LIN {X 0,Y 121.396,Z 550.061,A -85,B 0,C 180,E1 -28958.912,E2 -28958.912} C_VEL
LIN {X 0,Y 125.101,Z 540.479,A -85,B 0,C 180,E1 -28959.728,E2 -28959.728} C_VEL
LIN {X 0,Y 128.467,Z 528.906,A -85,B 0,C 180,E1 -28960.451,E2 -28960.451} C_VEL
LIN {X 0,Y 130.512,Z 518.787,A -85,B 0,C 180,E1 -28960.945,E2 -28960.945} C_VEL
LIN {X 0,Y 131.692,Z 509.827,A -85,B 0,C 180,E1 -28961.323,E2 -28961.323} C_VEL
LIN {X 0,Y 131.03,Z 507.265,A -85,B 0,C 180,E1 -28962.639,E2 -28962.639} C_VEL
LIN {X 0,Y 129.296,Z 502.882,A -85,B 0,C 180,E1 -28966.213,E2 -28966.213} C_VEL
LIN {X 0,Y 128.177,Z 500.193,A -85,B 0,C 180,E1 -28969.134,E2 -28969.134} C_VEL
LIN {X 0,Y 127.295,Z 497.903,A -85,B 0,C 180,E1 -28972.264,E2 -28972.264} C_VEL
LIN {X 0,Y 126.517,Z 494.337,A -85,B 0,C 180,E1 -28979.998,E2 -28979.998} C_VEL
LIN {X 0,Y 126.503,Z 495.032,A -85,B 0,C 180,E1 -28982.137,E2 -28982.137} C_VEL
LIN {X 0,Y 127.602,Z 498.617,A -85,B 0,C 180,E1 -28989.309,E2 -28989.309} C_VEL
LIN {X 0,Y 129.088,Z 502.368,A -85,B 0,C 180,E1 -28993.678,E2 -28993.678} C_VEL
LIN {X 0,Y 130.788,Z 506.608,A -85,B 0,C 180,E1 -28997.289,E2 -28997.289} C_VEL
LIN {X 0,Y 132.702,Z 512.359,A -85,B 0,C 180,E1 -29000.842,E2 -29000.842} C_VEL
LIN {X 0,Y 134.653,Z 519.518,A -85,B 0,C 180,E1 -29004.267,E2 -29004.267} C_VEL
LIN {X 0,Y 135.64,Z 526.664,A -85,B 0,C 180,E1 -29006.958,E2 -29006.958} C_VEL
LIN {X 0,Y 136.305,Z 538.938,A -85,B 0,C 180,E1 -29011.036,E2 -29011.036} C_VEL
LIN {X 0,Y 136.9,Z 550.921,A -85,B 0,C 180,E1 -29015.725,E2 -29015.725} C_VEL
LIN {X 0,Y 137.871,Z 560.467,A -85,B 0,C 180,E1 -29020.126,E2 -29020.126} C_VEL
LIN {X 0,Y 139.225,Z 567.985,A -85,B 0,C 180,E1 -29024.061,E2 -29024.061} C_VEL
LIN {X 0,Y 141.373,Z 575.718,A -85,B 0,C 180,E1 -29028.605,E2 -29028.605} C_VEL
LIN {X 0,Y 141.944,Z 579.169,A -85,B 0,C 180,E1 -29030.582,E2 -29030.582} C_VEL
LIN {X 0,Y 141.721,Z 585.194,A -85,B 0,C 180,E1 -29033.799,E2 -29033.799} C_VEL
LIN {X 0,Y 142.042,Z 590.615,A -85,B 0,C 180,E1 -29037.097,E2 -29037.097} C_VEL
LIN {X 0,Y 143.437,Z 593.097,A -85,B 0,C 180,E1 -29039.116,E2 -29039.116} C_VEL
LIN {X 0,Y 148.818,Z 598.103,A -85,B 0,C 180,E1 -29043.799,E2 -29043.799} C_VEL
LIN {X 0,Y 156.674,Z 603.043,A -85,B 0,C 180,E1 -29048.969,E2 -29048.969} C_VEL
LIN {X 0,Y 163.45,Z 606.067,A -85,B 0,C 180,E1 -29052.483,E2 -29052.483} C_VEL
LIN {X 0,Y 173.347,Z 609.238,A -85,B 0,C 180,E1 -29056.657,E2 -29056.657} C_VEL
LIN {X 0,Y 187.7,Z 612.106,A -85,B 0,C 180,E1 -29061.386,E2 -29061.386} C_VEL
LIN {X 0,Y 197.793,Z 613.431,A -85,B 0,C 180,E1 -29064.197,E2 -29064.197} C_VEL
LIN {X 0,Y 204.875,Z 614,A -85,B 0,C 180,E1 -29066.065,E2 -29066.065} C_VEL
LIN {X 0,Y 212.438,Z 614.386,A -85,B 0,C 180,E1 -29068.104,E2 -29068.104} C_VEL
LIN {X 0,Y 218.12,Z 614.456,A -85,B 0,C 180,E1 -29069.999,E2 -29069.999} C_VEL
LIN {X 0,Y 211.005,Z 614.354,A -85,B 0,C 180,E1 -29072.297,E2 -29072.297} C_VEL
LIN {X 0,Y 204.327,Z 613.955,A -85,B 0,C 180,E1 -29074.086,E2 -29074.086} C_VEL
LIN {X 0,Y 191.41,Z 612.636,A -85,B 0,C 180,E1 -29077.548,E2 -29077.548} C_VEL
LIN {X 0,Y 179.043,Z 610.552,A -85,B 0,C 180,E1 -29081.318,E2 -29081.318} C_VEL
LIN {X 0,Y 167.787,Z 607.605,A -85,B 0,C 180,E1 -29085.557,E2 -29085.557} C_VEL
LIN {X 0,Y 157.576,Z 603.516,A -85,B 0,C 180,E1 -29090.514,E2 -29090.514} C_VEL
LIN {X 0,Y 150.744,Z 599.534,A -85,B 0,C 180,E1 -29094.808,E2 -29094.808} C_VEL
LIN {X 0,Y 145.102,Z 594.893,A -85,B 0,C 180,E1 -29099.332,E2 -29099.332} C_VEL
LIN {X 0,Y 139.612,Z 588.206,A -85,B 0,C 180,E1 -29105.113,E2 -29105.113} C_VEL
LIN {X 0,Y 136.094,Z 581.344,A -85,B 0,C 180,E1 -29110.389,E2 -29110.389} C_VEL
LIN {X 0,Y 133.867,Z 573.78,A -85,B 0,C 180,E1 -29115.49,E2 -29115.49} C_VEL
LIN {X 0,Y 132.559,Z 565.283,A -85,B 0,C 180,E1 -29120.492,E2 -29120.492} C_VEL
LIN {X 0,Y 132.044,Z 555.828,A -85,B 0,C 180,E1 -29125.25,E2 -29125.25} C_VEL
LIN {X 0,Y 132.018,Z 547.218,A -85,B 0,C 180,E1 -29129.003,E2 -29129.003} C_VEL
LIN {X 0,Y 132.156,Z 536.997,A -85,B 0,C 180,E1 -29132.829,E2 -29132.829} C_VEL
LIN {X 0,Y 131.94,Z 527.432,A -85,B 0,C 180,E1 -29136.247,E2 -29136.247} C_VEL
LIN {X 0,Y 131.085,Z 521.305,A -85,B 0,C 180,E1 -29138.991,E2 -29138.991} C_VEL
LIN {X 0,Y 129.805,Z 515.544,A -85,B 0,C 180,E1 -29142.169,E2 -29142.169} C_VEL
LIN {X 0,Y 128.332,Z 510.701,A -85,B 0,C 180,E1 -29145.735,E2 -29145.735} C_VEL
LIN {X 0,Y 127.024,Z 507.083,A -85,B 0,C 180,E1 -29149.441,E2 -29149.441} C_VEL
LIN {X 0,Y 126.276,Z 504.86,A -85,B 0,C 180,E1 -29152.406,E2 -29152.406} C_VEL
LIN {X 0,Y 125.651,Z 501.387,A -85,B 0,C 180,E1 -29160.002,E2 -29160.002} C_VEL
LIN {X 0,Y 126.497,Z 505.489,A -85,B 0,C 180,E1 -29168.187,E2 -29168.187} C_VEL
LIN {X 0,Y 127.745,Z 509.003,A -85,B 0,C 180,E1 -29172.311,E2 -29172.311} C_VEL
LIN {X 0,Y 129.118,Z 513.003,A -85,B 0,C 180,E1 -29175.693,E2 -29175.693} C_VEL
LIN {X 0,Y 129.183,Z 513.202,A -85,B 0,C 180,E1 -29175.841,E2 -29175.841} C_VEL
LIN {X 0,Y 127.004,Z 525.493,A -85,B 0,C 180,E1 -29176.327,E2 -29176.327} C_VEL
LIN {X 0,Y 124.313,Z 535.644,A -85,B 0,C 180,E1 -29176.865,E2 -29176.865} C_VEL
LIN {X 0,Y 121.073,Z 544.914,A -85,B 0,C 180,E1 -29177.487,E2 -29177.487} C_VEL
LIN {X 0,Y 116.651,Z 554.944,A -85,B 0,C 180,E1 -29178.4,E2 -29178.4} C_VEL
LIN {X 0,Y 111.805,Z 563.937,A -85,B 0,C 180,E1 -29179.462,E2 -29179.462} C_VEL
LIN {X 0,Y 106.248,Z 572.658,A -85,B 0,C 180,E1 -29180.885,E2 -29180.885} C_VEL
LIN {X 0,Y 100.761,Z 580.073,A -85,B 0,C 180,E1 -29182.46,E2 -29182.46} C_VEL
LIN {X 0,Y 93.078,Z 588.861,A -85,B 0,C 180,E1 -29185.035,E2 -29185.035} C_VEL
LIN {X 0,Y 87.114,Z 594.847,A -85,B 0,C 180,E1 -29187.451,E2 -29187.451} C_VEL
LIN {X 0,Y 79.925,Z 601.155,A -85,B 0,C 180,E1 -29190.985,E2 -29190.985} C_VEL
LIN {X 0,Y 72.35,Z 606.999,A -85,B 0,C 180,E1 -29195.882,E2 -29195.882} C_VEL
LIN {X 0,Y 65.679,Z 611.527,A -85,B 0,C 180,E1 -29201.497,E2 -29201.497} C_VEL
LIN {X 0,Y 59.09,Z 615.494,A -85,B 0,C 180,E1 -29209.148,E2 -29209.148} C_VEL
LIN {X 0,Y 53.751,Z 618.435,A -85,B 0,C 180,E1 -29218.469,E2 -29218.469} C_VEL
LIN {X 0,Y 51.177,Z 619.945,A -85,B 0,C 180,E1 -29225.673,E2 -29225.673} C_VEL
LIN {X 0,Y 48.488,Z 621.489,A -85,B 0,C 180,E1 -29241.669,E2 -29241.669} C_VEL
LIN {X 0,Y 48.376,Z 621.777,A -85,B 0,C 180,E1 -29250.002,E2 -29250.002} C_VEL
LIN {X 0,Y 49.39,Z 620.882,A -85,B 0,C 180,E1 -29266.537,E2 -29266.537} C_VEL
LIN {X 0,Y 51.173,Z 619.944,A -85,B 0,C 180,E1 -29274.334,E2 -29274.334} C_VEL
LIN {X 0,Y 57.139,Z 616.583,A -85,B 0,C 180,E1 -29287.953,E2 -29287.953} C_VEL
LIN {X 0,Y 63.354,Z 612.953,A -85,B 0,C 180,E1 -29296.144,E2 -29296.144} C_VEL
LIN {X 0,Y 70.653,Z 608.222,A -85,B 0,C 180,E1 -29302.73,E2 -29302.73} C_VEL
LIN {X 0,Y 77.206,Z 603.34,A -85,B 0,C 180,E1 -29307.356,E2 -29307.356} C_VEL
LIN {X 0,Y 84.22,Z 597.467,A -85,B 0,C 180,E1 -29311.19,E2 -29311.19} C_VEL
LIN {X 0,Y 90.09,Z 591.978,A -85,B 0,C 180,E1 -29313.784,E2 -29313.784} C_VEL
LIN {X 0,Y 97.683,Z 583.767,A -85,B 0,C 180,E1 -29316.54,E2 -29316.54} C_VEL
LIN {X 0,Y 103.895,Z 575.946,A -85,B 0,C 180,E1 -29318.454,E2 -29318.454} C_VEL
LIN {X 0,Y 109.432,Z 567.868,A -85,B 0,C 180,E1 -29319.928,E2 -29319.928} C_VEL
LIN {X 0,Y 115.037,Z 558.114,A -85,B 0,C 180,E1 -29321.255,E2 -29321.255} C_VEL
LIN {X 0,Y 119.672,Z 548.3,A -85,B 0,C 180,E1 -29322.234,E2 -29322.234} C_VEL
LIN {X 0,Y 123.406,Z 538.456,A -85,B 0,C 180,E1 -29322.959,E2 -29322.959} C_VEL
LIN {X 0,Y 126.258,Z 528.753,A -85,B 0,C 180,E1 -29323.487,E2 -29323.487} C_VEL
LIN {X 0,Y 128.401,Z 518.416,A -85,B 0,C 180,E1 -29323.94,E2 -29323.94} C_VEL
LIN {X 0,Y 129.146,Z 513.097,A -85,B 0,C 180,E1 -29324.209,E2 -29324.209} C_VEL
LIN {X 0,Y 127.817,Z 509.204,A -85,B 0,C 180,E1 -29327.494,E2 -29327.494} C_VEL
LIN {X 0,Y 126.593,Z 505.776,A -85,B 0,C 180,E1 -29331.418,E2 -29331.418} C_VEL
LIN {X 0,Y 126.106,Z 504.468,A -85,B 0,C 180,E1 -29333.599,E2 -29333.599} C_VEL
LIN {X 0,Y 125.649,Z 501.401,A -85,B 0,C 180,E1 -29339.998,E2 -29339.998} C_VEL
LIN {X 0,Y 126.455,Z 505.345,A -85,B 0,C 180,E1 -29348.387,E2 -29348.387} C_VEL
LIN {X 0,Y 127.749,Z 509.022,A -85,B 0,C 180,E1 -29352.71,E2 -29352.71} C_VEL
LIN {X 0,Y 129.149,Z 513.386,A -85,B 0,C 180,E1 -29356.395,E2 -29356.395} C_VEL
LIN {X 0,Y 130.715,Z 519.225,A -85,B 0,C 180,E1 -29359.941,E2 -29359.941} C_VEL
LIN {X 0,Y 131.733,Z 525.753,A -85,B 0,C 180,E1 -29363.064,E2 -29363.064} C_VEL
LIN {X 0,Y 132.16,Z 531.637,A -85,B 0,C 180,E1 -29365.307,E2 -29365.307} C_VEL
LIN {X 0,Y 132.044,Z 542.178,A -85,B 0,C 180,E1 -29369.019,E2 -29369.019} C_VEL
LIN {X 0,Y 131.987,Z 551.545,A -85,B 0,C 180,E1 -29372.818,E2 -29372.818} C_VEL
LIN {X 0,Y 132.259,Z 560.714,A -85,B 0,C 180,E1 -29377.148,E2 -29377.148} C_VEL
LIN {X 0,Y 133.064,Z 569.328,A -85,B 0,C 180,E1 -29381.831,E2 -29381.831} C_VEL
LIN {X 0,Y 134.742,Z 577.422,A -85,B 0,C 180,E1 -29386.903,E2 -29386.903} C_VEL
LIN {X 0,Y 137.634,Z 584.788,A -85,B 0,C 180,E1 -29392.21,E2 -29392.21} C_VEL
LIN {X 0,Y 141.773,Z 591.188,A -85,B 0,C 180,E1 -29397.426,E2 -29397.426} C_VEL
LIN {X 0,Y 143.437,Z 593.097,A -85,B 0,C 180,E1 -29399.116,E2 -29399.116} C_VEL
LIN {X 0,Y 145.006,Z 595.651,A -85,B 0,C 180,E1 -29401.16,E2 -29401.16} C_VEL
LIN {X 0,Y 146.358,Z 599.989,A -85,B 0,C 180,E1 -29404.628,E2 -29404.628} C_VEL
LIN {X 0,Y 148.28,Z 603.811,A -85,B 0,C 180,E1 -29408.084,E2 -29408.084} C_VEL
LIN {X 0,Y 150.685,Z 605.496,A -85,B 0,C 180,E1 -29410.034,E2 -29410.034} C_VEL
LIN {X 0,Y 160.153,Z 609.047,A -85,B 0,C 180,E1 -29414.884,E2 -29414.884} C_VEL
LIN {X 0,Y 171.609,Z 611.758,A -85,B 0,C 180,E1 -29419.377,E2 -29419.377} C_VEL
LIN {X 0,Y 184.654,Z 613.614,A -85,B 0,C 180,E1 -29423.443,E2 -29423.443} C_VEL
LIN {X 0,Y 197.092,Z 614.548,A -85,B 0,C 180,E1 -29426.771,E2 -29426.771} C_VEL
LIN {X 0,Y 203.874,Z 614.693,A -85,B 0,C 180,E1 -29428.533,E2 -29428.533} C_VEL
LIN {X 0,Y 208.936,Z 614.708,A -85,B 0,C 180,E1 -29429.999,E2 -29429.999} C_VEL
LIN {X 0,Y 201.841,Z 614.672,A -85,B 0,C 180,E1 -29431.995,E2 -29431.995} C_VEL
LIN {X 0,Y 190.462,Z 614.094,A -85,B 0,C 180,E1 -29434.95,E2 -29434.95} C_VEL
LIN {X 0,Y 175.802,Z 612.432,A -85,B 0,C 180,E1 -29439.201,E2 -29439.201} C_VEL
LIN {X 0,Y 165.738,Z 610.468,A -85,B 0,C 180,E1 -29442.769,E2 -29442.769} C_VEL
LIN {X 0,Y 159.766,Z 608.917,A -85,B 0,C 180,E1 -29445.303,E2 -29445.303} C_VEL
LIN {X 0,Y 149.948,Z 605.196,A -85,B 0,C 180,E1 -29450.387,E2 -29450.387} C_VEL
LIN {X 0,Y 141.156,Z 599.819,A -85,B 0,C 180,E1 -29456.62,E2 -29456.62} C_VEL
LIN {X 0,Y 135.812,Z 594.731,A -85,B 0,C 180,E1 -29461.873,E2 -29461.873} C_VEL
LIN {X 0,Y 131.364,Z 588.149,A -85,B 0,C 180,E1 -29467.9,E2 -29467.9} C_VEL
LIN {X 0,Y 128.897,Z 581.531,A -85,B 0,C 180,E1 -29473.216,E2 -29473.216} C_VEL
LIN {X 0,Y 127.492,Z 573.853,A -85,B 0,C 180,E1 -29478.588,E2 -29478.588} C_VEL
LIN {X 0,Y 127.054,Z 565.701,A -85,B 0,C 180,E1 -29483.517,E2 -29483.517} C_VEL
LIN {X 0,Y 127.255,Z 556.153,A -85,B 0,C 180,E1 -29488.45,E2 -29488.45} C_VEL
LIN {X 0,Y 127.846,Z 547.744,A -85,B 0,C 180,E1 -29492.143,E2 -29492.143} C_VEL
LIN {X 0,Y 128.544,Z 536.897,A -85,B 0,C 180,E1 -29496.286,E2 -29496.286} C_VEL
LIN {X 0,Y 128.614,Z 529.501,A -85,B 0,C 180,E1 -29499.26,E2 -29499.26} C_VEL
LIN {X 0,Y 127.783,Z 522.727,A -85,B 0,C 180,E1 -29502.807,E2 -29502.807} C_VEL
LIN {X 0,Y 126.864,Z 517.935,A -85,B 0,C 180,E1 -29506.18,E2 -29506.18} C_VEL
LIN {X 0,Y 125.793,Z 513.912,A -85,B 0,C 180,E1 -29510.15,E2 -29510.15} C_VEL
LIN {X 0,Y 125.189,Z 511.697,A -85,B 0,C 180,E1 -29513.15,E2 -29513.15} C_VEL
LIN {X 0,Y 124.763,Z 508.615,A -85,B 0,C 180,E1 -29520.002,E2 -29520.002} C_VEL
LIN {X 0,Y 125.386,Z 512.335,A -85,B 0,C 180,E1 -29527.449,E2 -29527.449} C_VEL
LIN {X 0,Y 126.184,Z 515.156,A -85,B 0,C 180,E1 -29530.836,E2 -29530.836} C_VEL
LIN {X 0,Y 126.77,Z 517.302,A -85,B 0,C 180,E1 -29532.887,E2 -29532.887} C_VEL
LIN {X 0,Y 124.279,Z 529.09,A -85,B 0,C 180,E1 -29533.363,E2 -29533.363} C_VEL
LIN {X 0,Y 120.216,Z 542.165,A -85,B 0,C 180,E1 -29534.09,E2 -29534.09} C_VEL
LIN {X 0,Y 115.44,Z 553.16,A -85,B 0,C 180,E1 -29534.886,E2 -29534.886} C_VEL
LIN {X 0,Y 109.644,Z 563.742,A -85,B 0,C 180,E1 -29535.962,E2 -29535.962} C_VEL
LIN {X 0,Y 103.922,Z 572.462,A -85,B 0,C 180,E1 -29537.214,E2 -29537.214} C_VEL
LIN {X 0,Y 98.26,Z 579.877,A -85,B 0,C 180,E1 -29538.618,E2 -29538.618} C_VEL
LIN {X 0,Y 90.299,Z 588.666,A -85,B 0,C 180,E1 -29540.944,E2 -29540.944} C_VEL
LIN {X 0,Y 84.073,Z 594.652,A -85,B 0,C 180,E1 -29543.148,E2 -29543.148} C_VEL
LIN {X 0,Y 76.503,Z 600.96,A -85,B 0,C 180,E1 -29546.408,E2 -29546.408} C_VEL
LIN {X 0,Y 69.381,Z 606.192,A -85,B 0,C 180,E1 -29550.433,E2 -29550.433} C_VEL
LIN {X 0,Y 61.199,Z 611.331,A -85,B 0,C 180,E1 -29556.503,E2 -29556.503} C_VEL
LIN {X 0,Y 53.899,Z 615.299,A -85,B 0,C 180,E1 -29564.184,E2 -29564.184} C_VEL
LIN {X 0,Y 47.811,Z 618.239,A -85,B 0,C 180,E1 -29573.99,E2 -29573.99} C_VEL
LIN {X 0,Y 44.769,Z 619.749,A -85,B 0,C 180,E1 -29581.907,E2 -29581.907} C_VEL
LIN {X 0,Y 41.459,Z 621.294,A -85,B 0,C 180,E1 -29600.243,E2 -29600.243} C_VEL
LIN {X 0,Y 41.29,Z 621.582,A -85,B 0,C 180,E1 -29610.003,E2 -29610.003} C_VEL
LIN {X 0,Y 42.608,Z 620.687,A -85,B 0,C 180,E1 -29629.265,E2 -29629.265} C_VEL
LIN {X 0,Y 44.766,Z 619.748,A -85,B 0,C 180,E1 -29638.101,E2 -29638.101} C_VEL
LIN {X 0,Y 51.716,Z 616.388,A -85,B 0,C 180,E1 -29652.806,E2 -29652.806} C_VEL
LIN {X 0,Y 58.633,Z 612.757,A -85,B 0,C 180,E1 -29661.182,E2 -29661.182} C_VEL
LIN {X 0,Y 63.872,Z 609.816,A -85,B 0,C 180,E1 -29665.615,E2 -29665.615} C_VEL
LIN {X 0,Y 72.168,Z 604.237,A -85,B 0,C 180,E1 -29671.22,E2 -29671.22} C_VEL
LIN {X 0,Y 79.51,Z 598.583,A -85,B 0,C 180,E1 -29674.962,E2 -29674.962} C_VEL
LIN {X 0,Y 87.18,Z 591.782,A -85,B 0,C 180,E1 -29677.984,E2 -29677.984} C_VEL
LIN {X 0,Y 95.067,Z 583.571,A -85,B 0,C 180,E1 -29680.489,E2 -29680.489} C_VEL
LIN {X 0,Y 101.496,Z 575.75,A -85,B 0,C 180,E1 -29682.197,E2 -29682.197} C_VEL
LIN {X 0,Y 107.202,Z 567.673,A -85,B 0,C 180,E1 -29683.496,E2 -29683.496} C_VEL
LIN {X 0,Y 112.96,Z 557.919,A -85,B 0,C 180,E1 -29684.659,E2 -29684.659} C_VEL
LIN {X 0,Y 117.577,Z 548.4,A -85,B 0,C 180,E1 -29685.503,E2 -29685.503} C_VEL
LIN {X 0,Y 121.516,Z 538.262,A -85,B 0,C 180,E1 -29686.159,E2 -29686.159} C_VEL
LIN {X 0,Y 124.51,Z 528.186,A -85,B 0,C 180,E1 -29686.649,E2 -29686.649} C_VEL
LIN {X 0,Y 126.623,Z 518.222,A -85,B 0,C 180,E1 -29687.024,E2 -29687.024} C_VEL
LIN {X 0,Y 126.716,Z 517.201,A -85,B 0,C 180,E1 -29687.18,E2 -29687.18} C_VEL
LIN {X 0,Y 125.644,Z 513.41,A -85,B 0,C 180,E1 -29691.15,E2 -29691.15} C_VEL
LIN {X 0,Y 125.139,Z 511.46,A -85,B 0,C 180,E1 -29693.954,E2 -29693.954} C_VEL
LIN {X 0,Y 124.76,Z 508.639,A -85,B 0,C 180,E1 -29699.998,E2 -29699.998} C_VEL
LIN {X 0,Y 124.815,Z 510.441,A -85,B 0,C 180,E1 -29704.034,E2 -29704.034} C_VEL
LIN {X 0,Y 125.304,Z 512.181,A -85,B 0,C 180,E1 -29707.653,E2 -29707.653} C_VEL
LIN {X 0,Y 126.24,Z 515.75,A -85,B 0,C 180,E1 -29711.845,E2 -29711.845} C_VEL
LIN {X 0,Y 127.352,Z 519.998,A -85,B 0,C 180,E1 -29715.4,E2 -29715.4} C_VEL
LIN {X 0,Y 128.252,Z 526.327,A -85,B 0,C 180,E1 -29719.193,E2 -29719.193} C_VEL
LIN {X 0,Y 128.657,Z 531.878,A -85,B 0,C 180,E1 -29721.776,E2 -29721.776} C_VEL
LIN {X 0,Y 128.387,Z 540.389,A -85,B 0,C 180,E1 -29724.972,E2 -29724.972} C_VEL
LIN {X 0,Y 127.61,Z 551.058,A -85,B 0,C 180,E1 -29729.258,E2 -29729.258} C_VEL
LIN {X 0,Y 127.076,Z 560.958,A -85,B 0,C 180,E1 -29733.944,E2 -29733.944} C_VEL
LIN {X 0,Y 127.129,Z 569.086,A -85,B 0,C 180,E1 -29738.454,E2 -29738.454} C_VEL
LIN {X 0,Y 128.003,Z 577.228,A -85,B 0,C 180,E1 -29743.724,E2 -29743.724} C_VEL
LIN {X 0,Y 130.022,Z 585.057,A -85,B 0,C 180,E1 -29749.561,E2 -29749.561} C_VEL
LIN {X 0,Y 133.288,Z 591.386,A -85,B 0,C 180,E1 -29755.004,E2 -29755.004} C_VEL
LIN {X 0,Y 137.729,Z 596.74,A -85,B 0,C 180,E1 -29760.163,E2 -29760.163} C_VEL
LIN {X 0,Y 143.325,Z 601.406,A -85,B 0,C 180,E1 -29765.111,E2 -29765.111} C_VEL
LIN {X 0,Y 150.685,Z 605.496,A -85,B 0,C 180,E1 -29770.034,E2 -29770.034} C_VEL
LIN {X 0,Y 153.316,Z 607.032,A -85,B 0,C 180,E1 -29771.953,E2 -29771.953} C_VEL
LIN {X 0,Y 156.604,Z 609.767,A -85,B 0,C 180,E1 -29775.277,E2 -29775.277} C_VEL
LIN {X 0,Y 160.498,Z 611.94,A -85,B 0,C 180,E1 -29778.455,E2 -29778.455} C_VEL
LIN {X 0,Y 163.967,Z 612.735,A -85,B 0,C 180,E1 -29780.097,E2 -29780.097} C_VEL
LIN {X 0,Y 176.614,Z 614.273,A -85,B 0,C 180,E1 -29784.154,E2 -29784.154} C_VEL
LIN {X 0,Y 190.609,Z 614.974,A -85,B 0,C 180,E1 -29787.886,E2 -29787.886} C_VEL
LIN {X 0,Y 198.987,Z 614.982,A -85,B 0,C 180,E1 -29789.999,E2 -29789.999} C_VEL
LIN {X 0,Y 189.904,Z 614.969,A -85,B 0,C 180,E1 -29792.297,E2 -29792.297} C_VEL
LIN {X 0,Y 172.647,Z 613.949,A -85,B 0,C 180,E1 -29797.014,E2 -29797.014} C_VEL
LIN {X 0,Y 156.09,Z 611.184,A -85,B 0,C 180,E1 -29803.009,E2 -29803.009} C_VEL
LIN {X 0,Y 147.219,Z 608.66,A -85,B 0,C 180,E1 -29807.304,E2 -29807.304} C_VEL
LIN {X 0,Y 137.829,Z 604.333,A -85,B 0,C 180,E1 -29813.394,E2 -29813.394} C_VEL
LIN {X 0,Y 131.933,Z 600.104,A -85,B 0,C 180,E1 -29818.647,E2 -29818.647} C_VEL
LIN {X 0,Y 127.375,Z 595.164,A -85,B 0,C 180,E1 -29824.147,E2 -29824.147} C_VEL
LIN {X 0,Y 123.763,Z 588.299,A -85,B 0,C 180,E1 -29830.779,E2 -29830.779} C_VEL
LIN {X 0,Y 122.161,Z 581.668,A -85,B 0,C 180,E1 -29836.344,E2 -29836.344} C_VEL
LIN {X 0,Y 121.616,Z 574.48,A -85,B 0,C 180,E1 -29841.598,E2 -29841.598} C_VEL
LIN {X 0,Y 122.026,Z 564.983,A -85,B 0,C 180,E1 -29847.414,E2 -29847.414} C_VEL
LIN {X 0,Y 122.941,Z 556.469,A -85,B 0,C 180,E1 -29851.852,E2 -29851.852} C_VEL
LIN {X 0,Y 124.298,Z 546.365,A -85,B 0,C 180,E1 -29856.245,E2 -29856.245} C_VEL
LIN {X 0,Y 125.349,Z 537.003,A -85,B 0,C 180,E1 -29859.929,E2 -29859.929} C_VEL
LIN {X 0,Y 125.444,Z 531.121,A -85,B 0,C 180,E1 -29862.813,E2 -29862.813} C_VEL
LIN {X 0,Y 124.981,Z 525.735,A -85,B 0,C 180,E1 -29866.175,E2 -29866.175} C_VEL
LIN {X 0,Y 124.408,Z 521.667,A -85,B 0,C 180,E1 -29869.834,E2 -29869.834} C_VEL
LIN {X 0,Y 123.881,Z 518.462,A -85,B 0,C 180,E1 -29873.896,E2 -29873.896} C_VEL
LIN {X 0,Y 123.698,Z 515.867,A -85,B 0,C 180,E1 -29880.002,E2 -29880.002} C_VEL
LIN {X 0,Y 123.986,Z 518.851,A -85,B 0,C 180,E1 -29886.307,E2 -29886.307} C_VEL
LIN {X 0,Y 124.566,Z 521.753,A -85,B 0,C 180,E1 -29889.859,E2 -29889.859} C_VEL
LIN {X 0,Y 121.448,Z 533.801,A -85,B 0,C 180,E1 -29890.348,E2 -29890.348} C_VEL
LIN {X 0,Y 117.676,Z 544.345,A -85,B 0,C 180,E1 -29890.887,E2 -29890.887} C_VEL
LIN {X 0,Y 112.974,Z 554.553,A -85,B 0,C 180,E1 -29891.548,E2 -29891.548} C_VEL
LIN {X 0,Y 107.91,Z 563.547,A -85,B 0,C 180,E1 -29892.341,E2 -29892.341} C_VEL
LIN {X 0,Y 102.048,Z 572.268,A -85,B 0,C 180,E1 -29893.407,E2 -29893.407} C_VEL
LIN {X 0,Y 96.225,Z 579.682,A -85,B 0,C 180,E1 -29894.6,E2 -29894.6} C_VEL
LIN {X 0,Y 88.01,Z 588.471,A -85,B 0,C 180,E1 -29896.622,E2 -29896.622} C_VEL
LIN {X 0,Y 81.535,Z 594.456,A -85,B 0,C 180,E1 -29898.537,E2 -29898.537} C_VEL
LIN {X 0,Y 73.603,Z 600.763,A -85,B 0,C 180,E1 -29901.418,E2 -29901.418} C_VEL
LIN {X 0,Y 65.38,Z 606.401,A -85,B 0,C 180,E1 -29905.47,E2 -29905.47} C_VEL
LIN {X 0,Y 57.255,Z 611.136,A -85,B 0,C 180,E1 -29910.773,E2 -29910.773} C_VEL
LIN {X 0,Y 49.198,Z 615.103,A -85,B 0,C 180,E1 -29918.221,E2 -29918.221} C_VEL
LIN {X 0,Y 42.247,Z 618.043,A -85,B 0,C 180,E1 -29928.29,E2 -29928.29} C_VEL
LIN {X 0,Y 38.626,Z 619.553,A -85,B 0,C 180,E1 -29936.921,E2 -29936.921} C_VEL
LIN {X 0,Y 34.479,Z 621.099,A -85,B 0,C 180,E1 -29958.243,E2 -29958.243} C_VEL
LIN {X 0,Y 34.179,Z 621.387,A -85,B 0,C 180,E1 -29970.003,E2 -29970.003} C_VEL
LIN {X 0,Y 35.968,Z 620.491,A -85,B 0,C 180,E1 -29993.007,E2 -29993.007} C_VEL
LIN {X 0,Y 38.624,Z 619.552,A -85,B 0,C 180,E1 -30003.088,E2 -30003.088} C_VEL
LIN {X 0,Y 46.73,Z 616.192,A -85,B 0,C 180,E1 -30018.766,E2 -30018.766} C_VEL
LIN {X 0,Y 54.448,Z 612.561,A -85,B 0,C 180,E1 -30027.037,E2 -30027.037} C_VEL
LIN {X 0,Y 60.129,Z 609.62,A -85,B 0,C 180,E1 -30031.24,E2 -30031.24} C_VEL
LIN {X 0,Y 69.009,Z 604.04,A -85,B 0,C 180,E1 -30036.434,E2 -30036.434} C_VEL
LIN {X 0,Y 76.77,Z 598.387,A -85,B 0,C 180,E1 -30039.779,E2 -30039.779} C_VEL
LIN {X 0,Y 84.773,Z 591.587,A -85,B 0,C 180,E1 -30042.441,E2 -30042.441} C_VEL
LIN {X 0,Y 92.93,Z 583.376,A -85,B 0,C 180,E1 -30044.633,E2 -30044.633} C_VEL
LIN {X 0,Y 99.549,Z 575.554,A -85,B 0,C 180,E1 -30046.105,E2 -30046.105} C_VEL
LIN {X 0,Y 105.401,Z 567.478,A -85,B 0,C 180,E1 -30047.208,E2 -30047.208} C_VEL
LIN {X 0,Y 111.295,Z 557.724,A -85,B 0,C 180,E1 -30048.179,E2 -30048.179} C_VEL
LIN {X 0,Y 115.869,Z 548.52,A -85,B 0,C 180,E1 -30048.878,E2 -30048.878} C_VEL
LIN {X 0,Y 119.792,Z 538.743,A -85,B 0,C 180,E1 -30049.413,E2 -30049.413} C_VEL
LIN {X 0,Y 122.865,Z 528.822,A -85,B 0,C 180,E1 -30049.827,E2 -30049.827} C_VEL
LIN {X 0,Y 124.573,Z 521.724,A -85,B 0,C 180,E1 -30050.142,E2 -30050.142} C_VEL
LIN {X 0,Y 123.893,Z 518.431,A -85,B 0,C 180,E1 -30054.301,E2 -30054.301} C_VEL
LIN {X 0,Y 123.654,Z 515.847,A -85,B 0,C 180,E1 -30059.998,E2 -30059.998} C_VEL
LIN {X 0,Y 123.636,Z 517.595,A -85,B 0,C 180,E1 -30064.073,E2 -30064.073} C_VEL
LIN {X 0,Y 123.963,Z 519.01,A -85,B 0,C 180,E1 -30066.918,E2 -30066.918} C_VEL
LIN {X 0,Y 124.533,Z 522.404,A -85,B 0,C 180,E1 -30070.978,E2 -30070.978} C_VEL
LIN {X 0,Y 125.093,Z 526.762,A -85,B 0,C 180,E1 -30074.539,E2 -30074.539} C_VEL
LIN {X 0,Y 125.441,Z 532.139,A -85,B 0,C 180,E1 -30077.74,E2 -30077.74} C_VEL
LIN {X 0,Y 125.332,Z 537.047,A -85,B 0,C 180,E1 -30080.07,E2 -30080.07} C_VEL
LIN {X 0,Y 124.556,Z 544.227,A -85,B 0,C 180,E1 -30082.896,E2 -30082.896} C_VEL
LIN {X 0,Y 123.576,Z 551.753,A -85,B 0,C 180,E1 -30085.999,E2 -30085.999} C_VEL
LIN {X 0,Y 122.39,Z 561.2,A -85,B 0,C 180,E1 -30090.531,E2 -30090.531} C_VEL
LIN {X 0,Y 121.735,Z 569.519,A -85,B 0,C 180,E1 -30095.26,E2 -30095.26} C_VEL
LIN {X 0,Y 121.745,Z 577.706,A -85,B 0,C 180,E1 -30100.709,E2 -30100.709} C_VEL
LIN {X 0,Y 122.863,Z 585.321,A -85,B 0,C 180,E1 -30106.652,E2 -30106.652} C_VEL
LIN {X 0,Y 124.981,Z 591.214,A -85,B 0,C 180,E1 -30111.926,E2 -30111.926} C_VEL
LIN {X 0,Y 128.773,Z 596.931,A -85,B 0,C 180,E1 -30117.766,E2 -30117.766} C_VEL
LIN {X 0,Y 133.846,Z 601.68,A -85,B 0,C 180,E1 -30123.203,E2 -30123.203} C_VEL
LIN {X 0,Y 142.34,Z 606.666,A -85,B 0,C 180,E1 -30129.78,E2 -30129.78} C_VEL
LIN {X 0,Y 148.781,Z 609.23,A -85,B 0,C 180,E1 -30133.535,E2 -30133.535} C_VEL
LIN {X 0,Y 158.15,Z 611.691,A -85,B 0,C 180,E1 -30137.857,E2 -30137.857} C_VEL
LIN {X 0,Y 163.967,Z 612.735,A -85,B 0,C 180,E1 -30140.097,E2 -30140.097} C_VEL
LIN {X 0,Y 167.608,Z 613.511,A -85,B 0,C 180,E1 -30141.685,E2 -30141.685} C_VEL
LIN {X 0,Y 172.607,Z 614.581,A -85,B 0,C 180,E1 -30144.545,E2 -30144.545} C_VEL
LIN {X 0,Y 176.804,Z 615.186,A -85,B 0,C 180,E1 -30146.746,E2 -30146.746} C_VEL
LIN {X 0,Y 180.68,Z 615.3,A -85,B 0,C 180,E1 -30148.175,E2 -30148.175} C_VEL
LIN {X 0,Y 182.17,Z 615.307,A -85,B 0,C 180,E1 -30148.581,E2 -30148.581} C_VEL
LIN {X 0,Y 187.878,Z 615.287,A -85,B 0,C 180,E1 -30149.999,E2 -30149.999} C_VEL
LIN {X 0,Y 175.94,Z 615.265,A -85,B 0,C 180,E1 -30153.018,E2 -30153.018} C_VEL
LIN {X 0,Y 160.856,Z 614.278,A -85,B 0,C 180,E1 -30157.531,E2 -30157.531} C_VEL
LIN {X 0,Y 150.578,Z 612.75,A -85,B 0,C 180,E1 -30161.445,E2 -30161.445} C_VEL
LIN {X 0,Y 138.213,Z 609.535,A -85,B 0,C 180,E1 -30167.763,E2 -30167.763} C_VEL
LIN {X 0,Y 128.321,Z 604.712,A -85,B 0,C 180,E1 -30175.149,E2 -30175.149} C_VEL
LIN {X 0,Y 122.955,Z 600.365,A -85,B 0,C 180,E1 -30180.979,E2 -30180.979} C_VEL
LIN {X 0,Y 118.562,Z 594.23,A -85,B 0,C 180,E1 -30188.129,E2 -30188.129} C_VEL
LIN {X 0,Y 116.677,Z 588.736,A -85,B 0,C 180,E1 -30193.716,E2 -30193.716} C_VEL
LIN {X 0,Y 115.867,Z 580.959,A -85,B 0,C 180,E1 -30200.445,E2 -30200.445} C_VEL
LIN {X 0,Y 116.304,Z 573.354,A -85,B 0,C 180,E1 -30206.019,E2 -30206.019} C_VEL
LIN {X 0,Y 117.354,Z 566.2,A -85,B 0,C 180,E1 -30210.508,E2 -30210.508} C_VEL
LIN {X 0,Y 119.215,Z 556.365,A -85,B 0,C 180,E1 -30215.63,E2 -30215.63} C_VEL
LIN {X 0,Y 121.05,Z 547.248,A -85,B 0,C 180,E1 -30219.615,E2 -30219.615} C_VEL
LIN {X 0,Y 122.325,Z 539.7,A -85,B 0,C 180,E1 -30222.805,E2 -30222.805} C_VEL
LIN {X 0,Y 122.553,Z 534.144,A -85,B 0,C 180,E1 -30225.896,E2 -30225.896} C_VEL
LIN {X 0,Y 122.54,Z 529.713,A -85,B 0,C 180,E1 -30229.259,E2 -30229.259} C_VEL
LIN {X 0,Y 122.229,Z 526.532,A -85,B 0,C 180,E1 -30232.776,E2 -30232.776} C_VEL
LIN {X 0,Y 122.135,Z 525.015,A -85,B 0,C 180,E1 -30235.05,E2 -30235.05} C_VEL
LIN {X 0,Y 122.27,Z 522.993,A -85,B 0,C 180,E1 -30240.002,E2 -30240.002} C_VEL
LIN {X 0,Y 122.272,Z 525.751,A -85,B 0,C 180,E1 -30245.775,E2 -30245.775} C_VEL
LIN {X 0,Y 122.338,Z 526.446,A -85,B 0,C 180,E1 -30246.753,E2 -30246.753} C_VEL
LIN {X 0,Y 119.839,Z 535.184,A -85,B 0,C 180,E1 -30247.086,E2 -30247.086} C_VEL
LIN {X 0,Y 116.23,Z 544.867,A -85,B 0,C 180,E1 -30247.492,E2 -30247.492} C_VEL
LIN {X 0,Y 111.77,Z 554.358,A -85,B 0,C 180,E1 -30247.979,E2 -30247.979} C_VEL
LIN {X 0,Y 106.618,Z 563.352,A -85,B 0,C 180,E1 -30248.611,E2 -30248.611} C_VEL
LIN {X 0,Y 100.642,Z 572.073,A -85,B 0,C 180,E1 -30249.481,E2 -30249.481} C_VEL
LIN {X 0,Y 94.684,Z 579.487,A -85,B 0,C 180,E1 -30250.436,E2 -30250.436} C_VEL
LIN {X 0,Y 86.244,Z 588.275,A -85,B 0,C 180,E1 -30252.086,E2 -30252.086} C_VEL
LIN {X 0,Y 79.555,Z 594.26,A -85,B 0,C 180,E1 -30253.659,E2 -30253.659} C_VEL
LIN {X 0,Y 71.31,Z 600.568,A -85,B 0,C 180,E1 -30256.081,E2 -30256.081} C_VEL
LIN {X 0,Y 63.281,Z 605.846,A -85,B 0,C 180,E1 -30259.282,E2 -30259.282} C_VEL
LIN {X 0,Y 53.962,Z 610.94,A -85,B 0,C 180,E1 -30264.268,E2 -30264.268} C_VEL
LIN {X 0,Y 45.137,Z 614.907,A -85,B 0,C 180,E1 -30271.095,E2 -30271.095} C_VEL
LIN {X 0,Y 37.223,Z 617.847,A -85,B 0,C 180,E1 -30280.96,E2 -30280.96} C_VEL
LIN {X 0,Y 32.889,Z 619.357,A -85,B 0,C 180,E1 -30290.134,E2 -30290.134} C_VEL
LIN {X 0,Y 27.547,Z 620.903,A -85,B 0,C 180,E1 -30315.224,E2 -30315.224} C_VEL
LIN {X 0,Y 27.071,Z 621.192,A -85,B 0,C 180,E1 -30330.004,E2 -30330.004} C_VEL
LIN {X 0,Y 29.531,Z 620.295,A -85,B 0,C 180,E1 -30358.427,E2 -30358.427} C_VEL
LIN {X 0,Y 32.888,Z 619.357,A -85,B 0,C 180,E1 -30369.877,E2 -30369.877} C_VEL
LIN {X 0,Y 42.369,Z 615.996,A -85,B 0,C 180,E1 -30386.039,E2 -30386.039} C_VEL
LIN {X 0,Y 50.925,Z 612.365,A -85,B 0,C 180,E1 -30393.775,E2 -30393.775} C_VEL
LIN {X 0,Y 57.038,Z 609.424,A -85,B 0,C 180,E1 -30397.54,E2 -30397.54} C_VEL
LIN {X 0,Y 66.478,Z 603.844,A -85,B 0,C 180,E1 -30402.081,E2 -30402.081} C_VEL
LIN {X 0,Y 74.605,Z 598.191,A -85,B 0,C 180,E1 -30404.927,E2 -30404.927} C_VEL
LIN {X 0,Y 82.906,Z 591.392,A -85,B 0,C 180,E1 -30407.129,E2 -30407.129} C_VEL
LIN {X 0,Y 91.303,Z 583.18,A -85,B 0,C 180,E1 -30408.942,E2 -30408.942} C_VEL
LIN {X 0,Y 98.085,Z 575.359,A -85,B 0,C 180,E1 -30410.138,E2 -30410.138} C_VEL
LIN {X 0,Y 104.058,Z 567.282,A -85,B 0,C 180,E1 -30411.028,E2 -30411.028} C_VEL
LIN {X 0,Y 110.062,Z 557.53,A -85,B 0,C 180,E1 -30411.792,E2 -30411.792} C_VEL
LIN {X 0,Y 114.539,Z 548.72,A -85,B 0,C 180,E1 -30412.336,E2 -30412.336} C_VEL
LIN {X 0,Y 118.928,Z 537.857,A -85,B 0,C 180,E1 -30412.812,E2 -30412.812} C_VEL
LIN {X 0,Y 121.961,Z 528.027,A -85,B 0,C 180,E1 -30413.137,E2 -30413.137} C_VEL
LIN {X 0,Y 122.332,Z 526.436,A -85,B 0,C 180,E1 -30413.279,E2 -30413.279} C_VEL
LIN {X 0,Y 122.184,Z 524.809,A -85,B 0,C 180,E1 -30415.875,E2 -30415.875} C_VEL
LIN {X 0,Y 122.277,Z 522.953,A -85,B 0,C 180,E1 -30420.41,E2 -30420.41} C_VEL
LIN {X 0,Y 122.187,Z 525.743,A -85,B 0,C 180,E1 -30426.189,E2 -30426.189} C_VEL
LIN {X 0,Y 122.485,Z 529.019,A -85,B 0,C 180,E1 -30430.119,E2 -30430.119} C_VEL
LIN {X 0,Y 122.575,Z 532.899,A -85,B 0,C 180,E1 -30433.257,E2 -30433.257} C_VEL
LIN {X 0,Y 122.385,Z 538.666,A -85,B 0,C 180,E1 -30436.684,E2 -30436.684} C_VEL
LIN {X 0,Y 121.527,Z 544.575,A -85,B 0,C 180,E1 -30439.313,E2 -30439.313} C_VEL
LIN {X 0,Y 119.831,Z 553.14,A -85,B 0,C 180,E1 -30442.861,E2 -30442.861} C_VEL
LIN {X 0,Y 117.976,Z 562.607,A -85,B 0,C 180,E1 -30447.53,E2 -30447.53} C_VEL
LIN {X 0,Y 116.796,Z 569.751,A -85,B 0,C 180,E1 -30451.661,E2 -30451.661} C_VEL
LIN {X 0,Y 115.935,Z 578.041,A -85,B 0,C 180,E1 -30457.313,E2 -30457.313} C_VEL
LIN {X 0,Y 116.174,Z 585.581,A -85,B 0,C 180,E1 -30463.452,E2 -30463.452} C_VEL
LIN {X 0,Y 117.409,Z 591.314,A -85,B 0,C 180,E1 -30468.817,E2 -30468.817} C_VEL
LIN {X 0,Y 120.191,Z 597.005,A -85,B 0,C 180,E1 -30474.945,E2 -30474.945} C_VEL
LIN {X 0,Y 124.581,Z 601.91,A -85,B 0,C 180,E1 -30480.967,E2 -30480.967} C_VEL
LIN {X 0,Y 132.226,Z 606.958,A -85,B 0,C 180,E1 -30488.157,E2 -30488.157} C_VEL
LIN {X 0,Y 139.583,Z 609.983,A -85,B 0,C 180,E1 -30493.061,E2 -30493.061} C_VEL
LIN {X 0,Y 152.532,Z 613.069,A -85,B 0,C 180,E1 -30499.379,E2 -30499.379} C_VEL
LIN {X 0,Y 162.813,Z 614.457,A -85,B 0,C 180,E1 -30503.117,E2 -30503.117} C_VEL
LIN {X 0,Y 178.902,Z 615.29,A -85,B 0,C 180,E1 -30507.748,E2 -30507.748} C_VEL
LIN {X 0,Y 182.17,Z 615.307,A -85,B 0,C 180,E1 -30508.581,E2 -30508.581} C_VEL
LIN {X 0,Y 181.106,Z 615.358,A -85,B 0,C 180,E1 -30508.697,E2 -30508.697} C_VEL
LIN {X 0,Y 175.455,Z 615.457,A -85,B 0,C 180,E1 -30508.213,E2 -30508.213} C_VEL
LIN {X 0,Y 163.567,Z 615.487,A -85,B 0,C 180,E1 -30506.169,E2 -30506.169} C_VEL
LIN {X 0,Y 156.313,Z 615.167,A -85,B 0,C 180,E1 -30504.377,E2 -30504.377} C_VEL
LIN {X 0,Y 154.104,Z 615.002,A -85,B 0,C 180,E1 -30503.664,E2 -30503.664} C_VEL
LIN {X 0,Y 143.026,Z 613.678,A -85,B 0,C 180,E1 -30499.335,E2 -30499.335} C_VEL
LIN {X 0,Y 134.114,Z 611.793,A -85,B 0,C 180,E1 -30494.81,E2 -30494.81} C_VEL
LIN {X 0,Y 127.031,Z 609.481,A -85,B 0,C 180,E1 -30490.135,E2 -30490.135} C_VEL
LIN {X 0,Y 118.813,Z 604.868,A -85,B 0,C 180,E1 -30482.529,E2 -30482.529} C_VEL
LIN {X 0,Y 114.349,Z 600.665,A -85,B 0,C 180,E1 -30476.416,E2 -30476.416} C_VEL
LIN {X 0,Y 111.235,Z 594.972,A -85,B 0,C 180,E1 -30469.3,E2 -30469.3} C_VEL
LIN {X 0,Y 110.086,Z 589.472,A -85,B 0,C 180,E1 -30463.333,E2 -30463.333} C_VEL
LIN {X 0,Y 110.265,Z 581.128,A -85,B 0,C 180,E1 -30455.814,E2 -30455.814} C_VEL
LIN {X 0,Y 111.569,Z 573.686,A -85,B 0,C 180,E1 -30450.258,E2 -30450.258} C_VEL
LIN {X 0,Y 113.563,Z 565.401,A -85,B 0,C 180,E1 -30445.073,E2 -30445.073} C_VEL
LIN {X 0,Y 116.222,Z 555.534,A -85,B 0,C 180,E1 -30440.026,E2 -30440.026} C_VEL
LIN {X 0,Y 118.486,Z 547.001,A -85,B 0,C 180,E1 -30436.362,E2 -30436.362} C_VEL
LIN {X 0,Y 119.537,Z 541.558,A -85,B 0,C 180,E1 -30433.6,E2 -30433.6} C_VEL
LIN {X 0,Y 119.909,Z 537.813,A -85,B 0,C 180,E1 -30431.155,E2 -30431.155} C_VEL
LIN {X 0,Y 120.077,Z 534.432,A -85,B 0,C 180,E1 -30428.091,E2 -30428.091} C_VEL
LIN {X 0,Y 120.142,Z 532.842,A -85,B 0,C 180,E1 -30426.035,E2 -30426.035} C_VEL
LIN {X 0,Y 120.248,Z 531.344,A -85,B 0,C 180,E1 -30423.349,E2 -30423.349} C_VEL
LIN {X 0,Y 120.453,Z 530.122,A -85,B 0,C 180,E1 -30419.789,E2 -30419.789} C_VEL
LIN {X 0,Y 120.328,Z 531.479,A -85,B 0,C 180,E1 -30416.65,E2 -30416.65} C_VEL
LIN {X 0,Y 119.723,Z 533.4,A -85,B 0,C 180,E1 -30416.32,E2 -30416.32} C_VEL
LIN {X 0,Y 115.514,Z 544.679,A -85,B 0,C 180,E1 -30416.014,E2 -30416.014} C_VEL
LIN {X 0,Y 111.011,Z 554.156,A -85,B 0,C 180,E1 -30415.653,E2 -30415.653} C_VEL
LIN {X 0,Y 105.795,Z 563.152,A -85,B 0,C 180,E1 -30415.176,E2 -30415.176} C_VEL
LIN {X 0,Y 99.721,Z 571.872,A -85,B 0,C 180,E1 -30414.556,E2 -30414.556} C_VEL
LIN {X 0,Y 93.665,Z 579.288,A -85,B 0,C 180,E1 -30413.824,E2 -30413.824} C_VEL
LIN {X 0,Y 85.049,Z 588.077,A -85,B 0,C 180,E1 -30412.583,E2 -30412.583} C_VEL
LIN {X 0,Y 78.191,Z 594.063,A -85,B 0,C 180,E1 -30411.386,E2 -30411.386} C_VEL
LIN {X 0,Y 69.687,Z 600.371,A -85,B 0,C 180,E1 -30409.518,E2 -30409.518} C_VEL
LIN {X 0,Y 60.984,Z 605.826,A -85,B 0,C 180,E1 -30406.864,E2 -30406.864} C_VEL
LIN {X 0,Y 51.452,Z 610.743,A -85,B 0,C 180,E1 -30402.976,E2 -30402.976} C_VEL
LIN {X 0,Y 41.905,Z 614.71,A -85,B 0,C 180,E1 -30397.289,E2 -30397.289} C_VEL
LIN {X 0,Y 32.989,Z 617.65,A -85,B 0,C 180,E1 -30388.455,E2 -30388.455} C_VEL
LIN {X 0,Y 27.791,Z 619.161,A -85,B 0,C 180,E1 -30379.353,E2 -30379.353} C_VEL
LIN {X 0,Y 20.748,Z 620.707,A -85,B 0,C 180,E1 -30349.805,E2 -30349.805} C_VEL
LIN {X 0,Y 19.977,Z 620.997,A -85,B 0,C 180,E1 -30330.006,E2 -30330.006} C_VEL
LIN {X 0,Y 23.513,Z 620.1,A -85,B 0,C 180,E1 -30293.295,E2 -30293.295} C_VEL
LIN {X 0,Y 27.79,Z 619.161,A -85,B 0,C 180,E1 -30280.659,E2 -30280.659} C_VEL
LIN {X 0,Y 38.839,Z 615.801,A -85,B 0,C 180,E1 -30265.217,E2 -30265.217} C_VEL
LIN {X 0,Y 48.204,Z 612.172,A -85,B 0,C 180,E1 -30258.624,E2 -30258.624} C_VEL
LIN {X 0,Y 54.701,Z 609.229,A -85,B 0,C 180,E1 -30255.517,E2 -30255.517} C_VEL
LIN {X 0,Y 64.632,Z 603.65,A -85,B 0,C 180,E1 -30251.873,E2 -30251.873} C_VEL
LIN {X 0,Y 73.068,Z 597.998,A -85,B 0,C 180,E1 -30249.65,E2 -30249.65} C_VEL
LIN {X 0,Y 81.606,Z 591.199,A -85,B 0,C 180,E1 -30247.965,E2 -30247.965} C_VEL
LIN {X 0,Y 90.201,Z 582.988,A -85,B 0,C 180,E1 -30246.595,E2 -30246.595} C_VEL
LIN {X 0,Y 97.117,Z 575.169,A -85,B 0,C 180,E1 -30245.729,E2 -30245.729} C_VEL
LIN {X 0,Y 103.189,Z 567.095,A -85,B 0,C 180,E1 -30245.099,E2 -30245.099} C_VEL
LIN {X 0,Y 109.271,Z 557.342,A -85,B 0,C 180,E1 -30244.527,E2 -30244.527} C_VEL
LIN {X 0,Y 113.597,Z 549.009,A -85,B 0,C 180,E1 -30244.143,E2 -30244.143} C_VEL
LIN {X 0,Y 117.888,Z 538.715,A -85,B 0,C 180,E1 -30243.817,E2 -30243.817} C_VEL
LIN {X 0,Y 119.715,Z 533.411,A -85,B 0,C 180,E1 -30243.65,E2 -30243.65} C_VEL
LIN {X 0,Y 120.316,Z 531.517,A -85,B 0,C 180,E1 -30243.351,E2 -30243.351} C_VEL
LIN {X 0,Y 120.476,Z 530.017,A -85,B 0,C 180,E1 -30240.002,E2 -30240.002} C_VEL
LIN {X 0,Y 120.255,Z 531.325,A -85,B 0,C 180,E1 -30236.651,E2 -30236.651} C_VEL
LIN {X 0,Y 120.128,Z 533.302,A -85,B 0,C 180,E1 -30233.282,E2 -30233.282} C_VEL
LIN {X 0,Y 119.992,Z 536.487,A -85,B 0,C 180,E1 -30229.882,E2 -30229.882} C_VEL
LIN {X 0,Y 119.707,Z 540.412,A -85,B 0,C 180,E1 -30227.099,E2 -30227.099} C_VEL
LIN {X 0,Y 118.929,Z 544.9,A -85,B 0,C 180,E1 -30224.58,E2 -30224.58} C_VEL
LIN {X 0,Y 117.018,Z 552.72,A -85,B 0,C 180,E1 -30221.215,E2 -30221.215} C_VEL
LIN {X 0,Y 114.564,Z 561.682,A -85,B 0,C 180,E1 -30216.949,E2 -30216.949} C_VEL
LIN {X 0,Y 112.477,Z 569.695,A -85,B 0,C 180,E1 -30212.381,E2 -30212.381} C_VEL
LIN {X 0,Y 110.607,Z 578.532,A -85,B 0,C 180,E1 -30206.254,E2 -30206.254} C_VEL
LIN {X 0,Y 109.94,Z 585.842,A -85,B 0,C 180,E1 -30200.092,E2 -30200.092} C_VEL
LIN {X 0,Y 110.353,Z 591.581,A -85,B 0,C 180,E1 -30194.469,E2 -30194.469} C_VEL
LIN {X 0,Y 112.159,Z 597.244,A -85,B 0,C 180,E1 -30188.026,E2 -30188.026} C_VEL
LIN {X 0,Y 116.712,Z 603.166,A -85,B 0,C 180,E1 -30180.03,E2 -30180.03} C_VEL
LIN {X 0,Y 122.626,Z 607.351,A -85,B 0,C 180,E1 -30173.514,E2 -30173.514} C_VEL
LIN {X 0,Y 127.869,Z 609.835,A -85,B 0,C 180,E1 -30169.254,E2 -30169.254} C_VEL
LIN {X 0,Y 137.302,Z 612.636,A -85,B 0,C 180,E1 -30163.466,E2 -30163.466} C_VEL
LIN {X 0,Y 149.209,Z 614.603,A -85,B 0,C 180,E1 -30158.122,E2 -30158.122} C_VEL
LIN {X 0,Y 161.998,Z 615.542,A -85,B 0,C 180,E1 -30153.812,E2 -30153.812} C_VEL
LIN {X 0,Y 176.286,Z 615.605,A -85,B 0,C 180,E1 -30149.999,E2 -30149.999} C_VEL
LIN {X 0,Y 157.806,Z 615.279,A -85,B 0,C 180,E1 -30144.889,E2 -30144.889} C_VEL
LIN {X 0,Y 154.104,Z 615.002,A -85,B 0,C 180,E1 -30143.664,E2 -30143.664} C_VEL
LIN {X 0,Y 149.422,Z 614.76,A -85,B 0,C 180,E1 -30142.306,E2 -30142.306} C_VEL
LIN {X 0,Y 133.964,Z 614.052,A -85,B 0,C 180,E1 -30138.71,E2 -30138.71} C_VEL
LIN {X 0,Y 129.501,Z 613.517,A -85,B 0,C 180,E1 -30137.058,E2 -30137.058} C_VEL
LIN {X 0,Y 128.24,Z 613.248,A -85,B 0,C 180,E1 -30136.399,E2 -30136.399} C_VEL
LIN {X 0,Y 117.86,Z 610.127,A -85,B 0,C 180,E1 -30129.035,E2 -30129.035} C_VEL
LIN {X 0,Y 111.303,Z 606.446,A -85,B 0,C 180,E1 -30122.125,E2 -30122.125} C_VEL
LIN {X 0,Y 106.163,Z 600.94,A -85,B 0,C 180,E1 -30113.43,E2 -30113.43} C_VEL
LIN {X 0,Y 104.216,Z 595.851,A -85,B 0,C 180,E1 -30106.549,E2 -30106.549} C_VEL
LIN {X 0,Y 103.939,Z 589.113,A -85,B 0,C 180,E1 -30098.983,E2 -30098.983} C_VEL
